C03656=1161.878,20.189,-47.884,-179.949,6.079,149.078
C03657=1161.873,20.439,-47.898,-179.947,6.081,149.077
C03658=1161.869,20.689,-47.912,-179.944,6.081,149.077
C03659=1161.864,20.939,-47.927,-179.941,6.082,149.076
C03660=1161.859,21.188,-47.941,-179.939,6.082,149.075
C03661=1161.854,21.437,-47.956,-179.936,6.083,149.075
C03662=1161.848,21.686,-47.970,-179.934,6.084,149.074
C03663=1161.843,21.936,-47.984,-179.931,6.085,149.074
C03664=1161.838,22.186,-47.999,-179.929,6.086,149.073
C03665=1161.833,22.436,-48.013,-179.926,6.086,149.072
C03666=1161.828,22.686,-48.028,-179.924,6.087,149.072
C03667=1161.823,22.935,-48.043,-179.921,6.088,149.071
C03668=1161.818,23.184,-48.057,-179.919,6.089,149.071
C03669=1161.813,23.433,-48.071,-179.916,6.090,149.070
C03670=1161.808,23.683,-48.085,-179.914,6.090,149.070
C03671=1161.803,23.933,-48.099,-179.911,6.092,149.069
C03672=1161.797,24.182,-48.115,-179.908,6.093,149.069
C03673=1161.792,24.432,-48.129,-179.906,6.093,149.068
C03674=1161.787,24.682,-48.144,-179.903,6.094,149.067
C03675=1161.783,24.931,-48.158,-179.900,6.095,149.067
C03676=1161.778,25.180,-48.173,-179.898,6.096,149.066
C03677=1161.773,25.430,-48.187,-179.896,6.097,149.066
C03678=1161.767,25.679,-48.202,-179.893,6.097,149.065
C03679=1161.762,25.928,-48.217,-179.891,6.098,149.064
C03680=1161.757,26.178,-48.231,-179.888,6.099,149.064
C03681=1161.752,26.428,-48.245,-179.885,6.100,149.063
C03682=1161.747,26.678,-48.259,-179.883,6.100,149.063
C03683=1161.742,26.927,-48.275,-179.881,6.101,149.062
C03684=1161.737,27.177,-48.289,-179.877,6.103,149.062
C03685=1161.732,27.426,-48.304,-179.875,6.103,149.061
C03686=1161.727,27.695,-48.319,-179.873,6.104,149.060
C03687=1161.721,27.964,-48.336,-179.869,6.105,149.060
C03688=1161.716,28.233,-48.351,-179.867,6.106,149.059
C03689=1161.711,28.502,-48.367,-179.864,6.107,149.059
C03690=1161.705,28.752,-48.382,-179.861,6.108,149.058
C03691=1161.700,29.000,-48.396,-179.859,6.109,149.057
C03692=1161.695,29.250,-48.411,-179.856,6.109,149.057
C03693=1161.690,29.499,-48.426,-179.854,6.111,149.056
C03694=1161.684,29.749,-48.441,-179.851,6.111,149.056
C03695=1161.680,29.998,-48.456,-179.849,6.112,149.055
C03696=1161.675,30.248,-48.470,-179.846,6.112,149.055
C03697=1161.669,30.497,-48.485,-179.843,6.114,149.054
C03698=1161.664,30.747,-48.500,-179.841,6.115,149.053
C03699=1161.659,30.997,-48.514,-179.839,6.115,149.053
C03700=1161.654,31.246,-48.530,-179.836,6.116,149.052
C03701=1161.649,31.496,-48.544,-179.833,6.118,149.052
C03702=1161.644,31.745,-48.559,-179.831,6.118,149.051
C03703=1161.639,31.995,-48.574,-179.828,6.119,149.051
C03704=1161.634,32.244,-48.589,-179.825,6.120,149.050
C03705=1161.629,32.493,-48.604,-179.823,6.121,149.049
C03706=1161.624,32.743,-48.619,-179.820,6.121,149.049
C03707=1161.619,32.992,-48.634,-179.818,6.122,149.048
C03708=1161.614,33.242,-48.648,-179.815,6.124,149.048
C03709=1161.609,33.492,-48.664,-179.812,6.124,149.047
C03710=1161.604,33.742,-48.678,-179.810,6.125,149.047
C03711=1161.599,33.991,-48.694,-179.807,6.126,149.046
C03712=1161.594,34.241,-48.708,-179.805,6.127,149.046
C03713=1161.589,34.490,-48.723,-179.802,6.128,149.045
C03714=1161.584,34.739,-48.739,-179.800,6.128,149.044
C03715=1161.579,34.989,-48.753,-179.797,6.130,149.044
C03716=1161.574,35.239,-48.768,-179.795,6.131,149.043
C03717=1161.569,35.488,-48.783,-179.792,6.131,149.043
C03718=1161.564,35.737,-48.798,-179.789,6.133,149.042
C03719=1161.559,35.987,-48.813,-179.787,6.133,149.041
C03720=1161.554,36.236,-48.828,-179.784,6.134,149.041
C03721=1161.548,36.486,-48.843,-179.782,6.134,149.040
C03722=1161.544,36.735,-48.858,-179.779,6.136,149.040
C03723=1161.538,36.984,-48.874,-179.776,6.137,149.039
C03724=1161.534,37.235,-48.888,-179.774,6.137,149.039
C03725=1161.529,37.484,-48.904,-179.771,6.139,149.038
C03726=1161.524,37.733,-48.919,-179.769,6.140,149.038
C03727=1161.518,37.983,-48.934,-179.766,6.140,149.037
C03728=1161.514,38.232,-48.949,-179.763,6.142,149.037
C03729=1161.508,38.482,-48.964,-179.761,6.142,149.036
C03730=1161.504,38.731,-48.979,-179.759,6.143,149.035
C03731=1161.498,38.981,-48.994,-179.755,6.144,149.035
C03732=1161.493,39.230,-49.009,-179.753,6.145,149.034
C03733=1161.488,39.480,-49.025,-179.751,6.146,149.034
C03734=1161.484,39.729,-49.040,-179.748,6.147,149.033
C03735=1161.478,39.979,-49.056,-179.745,6.148,149.033
C03736=1161.473,40.229,-49.071,-179.743,6.149,149.032
C03737=1161.468,40.478,-49.086,-179.740,6.150,149.031
C03738=1161.463,40.727,-49.101,-179.738,6.151,149.031
C03739=1161.458,40.976,-49.116,-179.735,6.151,149.030
C03740=1161.453,41.226,-49.132,-179.732,6.153,149.030
C03741=1161.449,41.475,-49.147,-179.730,6.153,149.029
C03742=1161.443,41.725,-49.162,-179.727,6.154,149.029
C03743=1161.438,41.975,-49.178,-179.724,6.156,149.028
C03744=1161.433,42.224,-49.193,-179.722,6.156,149.028
C03745=1161.428,42.474,-49.209,-179.719,6.157,149.027
C03746=1161.423,42.723,-49.224,-179.717,6.159,149.026
C03747=1161.418,42.972,-49.239,-179.714,6.159,149.026
C03748=1161.413,43.222,-49.255,-179.712,6.160,149.025
C03749=1161.408,43.471,-49.270,-179.709,6.161,149.025
C03750=1161.403,43.721,-49.286,-179.706,6.162,149.024
C03751=1161.398,43.970,-49.301,-179.704,6.163,149.024
C03752=1161.393,44.220,-49.316,-179.701,6.164,149.023
C03753=1161.388,44.469,-49.332,-179.698,6.165,149.022
C03754=1161.382,44.718,-49.347,-179.696,6.166,149.022
C03755=1161.378,44.968,-49.363,-179.693,6.167,149.021
C03756=1161.373,45.218,-49.378,-179.691,6.168,149.021
C03757=1161.368,45.467,-49.394,-179.688,6.168,149.020
C03758=1161.363,45.716,-49.409,-179.686,6.170,149.020
C03759=1161.358,45.966,-49.425,-179.683,6.171,149.019
C03760=1161.353,46.216,-49.441,-179.680,6.172,149.019
C03761=1161.348,46.465,-49.456,-179.678,6.173,149.018
C03762=1161.343,46.714,-49.471,-179.675,6.173,149.018
C03763=1161.338,46.964,-49.487,-179.673,6.175,149.017
C03764=1161.333,47.214,-49.503,-179.670,6.175,149.016
C03765=1161.328,47.463,-49.518,-179.668,6.176,149.016
C03766=1161.323,47.712,-49.533,-179.665,6.178,149.015
C03767=1161.318,47.962,-49.549,-179.662,6.178,149.015
C03768=1161.312,48.212,-49.565,-179.659,6.180,149.014
C03769=1161.308,48.461,-49.580,-179.657,6.181,149.014
C03770=1161.303,48.710,-49.596,-179.654,6.181,149.013
C03771=1161.298,48.960,-49.612,-179.652,6.183,149.013
C03772=1161.292,49.209,-49.628,-179.649,6.183,149.012
C03773=1161.288,49.459,-49.643,-179.647,6.184,149.012
C03774=1161.283,49.708,-49.659,-179.644,6.185,149.011
C03775=1161.278,49.958,-49.674,-179.641,6.186,149.010
C03776=1161.273,50.207,-49.691,-179.638,6.188,149.010
C03777=1161.268,50.456,-49.706,-179.636,6.188,149.009
C03778=1161.263,50.706,-49.721,-179.633,6.189,149.009
C03779=1161.258,50.956,-49.737,-179.631,6.191,149.008
C03780=1161.253,51.205,-49.753,-179.629,6.191,149.008
C03781=1161.248,51.454,-49.769,-179.625,6.193,149.007
C03782=1161.243,51.704,-49.785,-179.623,6.194,149.007
C03783=1161.238,51.953,-49.801,-179.620,6.194,149.006
C03784=1161.233,52.202,-49.816,-179.618,6.196,149.006
C03785=1161.229,52.452,-49.832,-179.615,6.196,149.005
C03786=1161.223,52.701,-49.848,-179.612,6.198,149.004
C03787=1161.218,52.951,-49.864,-179.610,6.198,149.004
C03788=1161.213,53.201,-49.880,-179.608,6.199,149.003
C03789=1161.208,53.450,-49.896,-179.604,6.201,149.003
C03790=1161.202,53.718,-49.913,-179.602,6.201,149.002
C03791=1161.197,53.987,-49.930,-179.599,6.203,149.002
C03792=1161.192,54.256,-49.947,-179.596,6.204,149.001
C03793=1161.186,54.524,-49.964,-179.594,6.205,149.000
C03794=1161.181,54.774,-49.980,-179.590,6.206,149.000
C03795=1161.176,55.023,-49.997,-179.588,6.207,148.999
C03796=1161.171,55.273,-50.012,-179.586,6.208,148.999
C03797=1161.167,55.522,-50.029,-179.583,6.209,148.998
C03798=1161.161,55.771,-50.044,-179.580,6.210,148.998
C03799=1161.156,56.021,-50.060,-179.577,6.211,148.997
C03800=1161.152,56.270,-50.076,-179.575,6.212,148.997
C03801=1161.147,56.519,-50.092,-179.572,6.213,148.996
C03802=1161.142,56.769,-50.108,-179.570,6.214,148.996
C03803=1161.137,57.018,-50.124,-179.567,6.215,148.995
C03804=1161.132,57.268,-50.140,-179.565,6.217,148.994
C03805=1161.127,57.517,-50.156,-179.562,6.217,148.994
C03806=1161.122,57.767,-50.172,-179.559,6.219,148.993
C03807=1161.117,58.016,-50.188,-179.557,6.219,148.993
C03808=1161.112,58.265,-50.204,-179.554,6.221,148.992
C03809=1161.106,58.515,-50.221,-179.552,6.222,148.992
C03810=1161.101,58.765,-50.237,-179.548,6.223,148.991
C03811=1161.097,59.014,-50.254,-179.546,6.224,148.991
C03812=1161.091,59.264,-50.269,-179.544,6.224,148.990
C03813=1161.087,59.513,-50.286,-179.541,6.226,148.990
C03814=1161.081,59.762,-50.301,-179.538,6.227,148.989
C03815=1161.077,60.012,-50.318,-179.535,6.228,148.989
C03816=1161.072,60.261,-50.334,-179.533,6.229,148.988
C03817=1161.067,60.511,-50.350,-179.530,6.230,148.987
C03818=1161.062,60.760,-50.367,-179.528,6.231,148.987
C03819=1161.057,61.010,-50.383,-179.525,6.233,148.986
C03820=1161.052,61.258,-50.399,-179.523,6.233,148.986
C03821=1161.048,61.508,-50.416,-179.519,6.235,148.985
C03822=1161.041,61.758,-50.432,-179.517,6.236,148.985
C03823=1161.037,62.007,-50.448,-179.514,6.237,148.984
C03824=1161.032,62.257,-50.464,-179.512,6.238,148.984
C03825=1161.027,62.506,-50.481,-179.510,6.239,148.983
C03826=1161.022,62.755,-50.497,-179.506,6.240,148.983
C03827=1161.017,63.005,-50.513,-179.504,6.241,148.982
C03828=1161.013,63.254,-50.530,-179.501,6.242,148.982
C03829=1161.008,63.503,-50.546,-179.499,6.243,148.981
C03830=1161.002,63.753,-50.563,-179.496,6.244,148.980
C03831=1160.997,64.002,-50.579,-179.494,6.245,148.980
C03832=1160.993,64.252,-50.595,-179.491,6.247,148.980
C03833=1160.987,64.501,-50.612,-179.488,6.247,148.979
C03834=1160.983,64.751,-50.628,-179.485,6.249,148.978
C03835=1160.977,65.001,-50.645,-179.483,6.250,148.978
C03836=1160.972,65.249,-50.661,-179.480,6.251,148.977
C03837=1160.968,65.499,-50.678,-179.477,6.252,148.977
C03838=1160.963,65.748,-50.693,-179.475,6.253,148.976
C03839=1160.958,65.998,-50.710,-179.473,6.254,148.976
C03840=1160.953,66.247,-50.727,-179.469,6.256,148.975
C03841=1160.948,66.496,-50.744,-179.467,6.256,148.975
C03842=1160.943,66.746,-50.760,-179.464,6.258,148.974
C03843=1160.938,66.995,-50.777,-179.462,6.259,148.974
C03844=1160.933,67.245,-50.793,-179.459,6.260,148.973
C03845=1160.928,67.494,-50.810,-179.456,6.261,148.973
C03846=1160.923,67.743,-50.826,-179.454,6.262,148.972
C03847=1160.919,67.993,-50.843,-179.451,6.263,148.971
C03848=1160.913,68.242,-50.860,-179.448,6.265,148.971
C03849=1160.908,68.491,-50.876,-179.446,6.265,148.970
C03850=1160.904,68.741,-50.893,-179.443,6.267,148.970
C03851=1160.898,68.990,-50.909,-179.441,6.268,148.970
C03852=1160.893,69.240,-50.926,-179.438,6.269,148.969
C03853=1160.889,69.489,-50.943,-179.435,6.270,148.968
C03854=1160.883,69.739,-50.960,-179.432,6.271,148.968
C03855=1160.878,69.988,-50.976,-179.430,6.272,148.967
C03856=1160.874,70.237,-50.993,-179.427,6.274,148.967
C03857=1160.868,70.487,-51.010,-179.425,6.274,148.966
C03858=1160.864,70.736,-51.026,-179.422,6.276,148.966
C03859=1160.859,70.986,-51.043,-179.419,6.277,148.965
C03860=1160.854,71.235,-51.060,-179.417,6.278,148.965
C03861=1160.849,71.484,-51.077,-179.414,6.280,148.964
C03862=1160.844,71.734,-51.093,-179.411,6.280,148.964
C03863=1160.839,71.983,-51.111,-179.408,6.282,148.963
C03864=1160.834,72.232,-51.127,-179.406,6.282,148.963
C03865=1160.829,72.482,-51.144,-179.403,6.284,148.962
C03866=1160.824,72.731,-51.161,-179.401,6.285,148.962
C03867=1160.819,72.980,-51.177,-179.398,6.286,148.961
C03868=1160.814,73.230,-51.194,-179.396,6.287,148.961
C03869=1160.810,73.480,-51.211,-179.392,6.289,148.960
C03870=1160.804,73.729,-51.228,-179.390,6.289,148.959
C03871=1160.800,73.977,-51.245,-179.387,6.291,148.959
C03872=1160.794,74.227,-51.263,-179.384,6.292,148.958
C03873=1160.790,74.477,-51.279,-179.382,6.293,148.958
C03874=1160.785,74.727,-51.297,-179.379,6.295,148.957
C03875=1160.780,74.975,-51.313,-179.377,6.295,148.957
C03876=1160.774,75.225,-51.330,-179.374,6.297,148.956
C03877=1160.770,75.475,-51.347,-179.371,6.298,148.956
C03878=1160.765,75.724,-51.364,-179.369,6.299,148.955
C03879=1160.760,75.973,-51.381,-179.367,6.300,148.955
C03880=1160.755,76.222,-51.398,-179.363,6.302,148.954
C03881=1160.750,76.472,-51.415,-179.361,6.303,148.954
C03882=1160.745,76.722,-51.432,-179.358,6.304,148.953
C03883=1160.741,76.971,-51.449,-179.355,6.305,148.953
C03884=1160.735,77.220,-51.467,-179.353,6.306,148.952
C03885=1160.731,77.469,-51.483,-179.350,6.308,148.952
C03886=1160.725,77.719,-51.501,-179.348,6.308,148.951
C03887=1160.721,77.968,-51.517,-179.345,6.310,148.951
C03888=1160.716,78.218,-51.535,-179.342,6.311,148.950
C03889=1160.711,78.466,-51.551,-179.340,6.312,148.950
C03890=1160.706,78.716,-51.569,-179.336,6.314,148.949
C03891=1160.701,78.965,-51.587,-179.334,6.315,148.949
C03892=1160.696,79.215,-51.603,-179.331,6.316,148.948
C03893=1160.691,79.465,-51.621,-179.329,6.317,148.948
C03894=1160.686,79.732,-51.638,-179.326,6.318,148.947
C03895=1160.681,80.001,-51.658,-179.323,6.320,148.947
C03896=1160.675,80.270,-51.676,-179.320,6.321,148.946
C03897=1160.670,80.537,-51.694,-179.317,6.323,148.945
C03898=1160.665,80.787,-51.711,-179.315,6.324,148.945
C03899=1160.660,81.036,-51.729,-179.312,6.325,148.944
C03900=1160.655,81.286,-51.746,-179.309,6.326,148.944
C03901=1160.651,81.535,-51.764,-179.307,6.328,148.944
C03902=1160.645,81.785,-51.781,-179.304,6.329,148.943
C03903=1160.641,82.034,-51.798,-179.301,6.330,148.942
C03904=1160.635,82.283,-51.816,-179.299,6.331,148.942
C03905=1160.630,82.533,-51.833,-179.296,6.332,148.941
C03906=1160.626,82.781,-51.850,-179.293,6.334,148.941
C03907=1160.621,83.031,-51.868,-179.291,6.335,148.941
C03908=1160.616,83.280,-51.886,-179.288,6.336,148.940
C03909=1160.611,83.530,-51.903,-179.285,6.338,148.939
C03910=1160.606,83.779,-51.920,-179.283,6.338,148.939
C03911=1160.601,84.029,-51.937,-179.280,6.340,148.938
C03912=1160.596,84.278,-51.955,-179.277,6.341,148.938
C03913=1160.592,84.528,-51.972,-179.274,6.342,148.937
C03914=1160.587,84.777,-51.990,-179.272,6.344,148.937
C03915=1160.582,85.027,-52.007,-179.269,6.345,148.936
C03916=1160.577,85.276,-52.025,-179.266,6.346,148.936
C03917=1160.572,85.524,-52.042,-179.264,6.348,148.935
C03918=1160.567,85.774,-52.060,-179.262,6.348,148.935
C03919=1160.562,86.023,-52.077,-179.258,6.350,148.934
C03920=1160.557,86.273,-52.095,-179.256,6.351,148.934
C03921=1160.552,86.522,-52.113,-179.253,6.352,148.933
C03922=1160.547,86.771,-52.129,-179.250,6.354,148.933
C03923=1160.542,87.020,-52.147,-179.247,6.355,148.932
C03924=1160.537,87.270,-52.165,-179.245,6.356,148.932
C03925=1160.532,87.519,-52.183,-179.242,6.358,148.931
C03926=1160.527,87.769,-52.201,-179.239,6.359,148.931
C03927=1160.523,88.018,-52.217,-179.237,6.360,148.930
C03928=1160.518,88.267,-52.235,-179.234,6.361,148.930
C03929=1160.513,88.516,-52.253,-179.231,6.363,148.929
C03930=1160.508,88.766,-52.271,-179.229,6.364,148.929
C03931=1160.503,89.015,-52.289,-179.226,6.365,148.928
C03932=1160.498,89.265,-52.307,-179.224,6.366,148.928
C03933=1160.493,89.514,-52.325,-179.221,6.368,148.928
C03934=1160.489,89.763,-52.341,-179.218,6.370,148.927
C03935=1160.484,90.012,-52.359,-179.216,6.370,148.926
C03936=1160.479,90.262,-52.377,-179.213,6.372,148.926
C03937=1160.474,90.511,-52.394,-179.210,6.374,148.926
C03938=1160.469,90.761,-52.412,-179.208,6.374,148.925
C03939=1160.464,91.010,-52.430,-179.205,6.376,148.925
C03940=1160.459,91.259,-52.448,-179.202,6.377,148.924
C03941=1160.454,91.509,-52.467,-179.200,6.378,148.923
C03942=1160.449,91.759,-52.484,-179.197,6.380,148.923
C03943=1160.444,92.008,-52.502,-179.194,6.381,148.923
C03944=1160.439,92.257,-52.520,-179.192,6.382,148.922
C03945=1160.435,92.506,-52.538,-179.189,6.384,148.922
C03946=1160.430,92.755,-52.556,-179.186,6.385,148.921
C03947=1160.425,93.004,-52.574,-179.183,6.386,148.920
C03948=1160.421,93.253,-52.591,-179.181,6.387,148.920
C03949=1160.415,93.503,-52.609,-179.178,6.389,148.920
C03950=1160.410,93.752,-52.627,-179.175,6.391,148.919
C03951=1160.405,94.001,-52.644,-179.173,6.391,148.919
C03952=1160.401,94.251,-52.662,-179.170,6.393,148.918
C03953=1160.396,94.501,-52.681,-179.167,6.395,148.918
C03954=1160.391,94.750,-52.699,-179.165,6.395,148.917
C03955=1160.386,94.999,-52.717,-179.162,6.397,148.917
C03956=1160.381,95.248,-52.735,-179.159,6.399,148.916
C03957=1160.376,95.498,-52.753,-179.156,6.399,148.916
C03958=1160.371,95.747,-52.771,-179.154,6.401,148.915
C03959=1160.366,95.996,-52.789,-179.151,6.403,148.915
C03960=1160.361,96.245,-52.807,-179.149,6.403,148.914
C03961=1160.357,96.495,-52.826,-179.146,6.405,148.914
C03962=1160.352,96.744,-52.844,-179.143,6.407,148.913
C03963=1160.347,96.993,-52.862,-179.140,6.408,148.913
C03964=1160.342,97.242,-52.880,-179.138,6.409,148.912
C03965=1160.337,97.492,-52.898,-179.135,6.410,148.912
C03966=1160.332,97.741,-52.916,-179.132,6.412,148.911
C03967=1160.328,97.991,-52.934,-179.130,6.413,148.911
C03968=1160.322,98.240,-52.952,-179.127,6.414,148.910
C03969=1160.317,98.489,-52.970,-179.124,6.416,148.910
C03970=1160.312,98.739,-52.988,-179.121,6.418,148.910
C03971=1160.308,98.988,-53.006,-179.119,6.418,148.909
C03972=1160.303,99.237,-53.024,-179.116,6.420,148.908
C03973=1160.299,99.486,-53.043,-179.113,6.422,148.908
C03974=1160.294,99.735,-53.061,-179.111,6.423,148.908
C03975=1160.288,99.985,-53.080,-179.108,6.424,148.907
C03976=1160.283,100.234,-53.098,-179.105,6.426,148.907
C03977=1160.279,100.484,-53.116,-179.102,6.427,148.906
C03978=1160.274,100.733,-53.134,-179.100,6.428,148.906
C03979=1160.269,100.982,-53.153,-179.097,6.430,148.905
C03980=1160.264,101.231,-53.172,-179.094,6.431,148.905
C03981=1160.259,101.480,-53.190,-179.092,6.433,148.904
C03982=1160.254,101.730,-53.208,-179.090,6.434,148.904
C03983=1160.250,101.979,-53.226,-179.086,6.435,148.903
C03984=1160.245,102.228,-53.245,-179.084,6.437,148.903
C03985=1160.239,102.477,-53.263,-179.081,6.439,148.902
C03986=1160.235,102.727,-53.281,-179.078,6.439,148.902
C03987=1160.230,102.976,-53.299,-179.076,6.441,148.901
C03988=1160.225,103.225,-53.318,-179.073,6.443,148.901
C03989=1160.220,103.475,-53.337,-179.070,6.444,148.901
C03990=1160.216,103.724,-53.355,-179.068,6.445,148.900
C03991=1160.211,103.973,-53.374,-179.065,6.446,148.899
C03992=1160.205,104.222,-53.392,-179.062,6.448,148.899
C03993=1160.201,104.472,-53.411,-179.059,6.450,148.899
C03994=1160.196,104.721,-53.429,-179.057,6.450,148.898
C03995=1160.191,104.970,-53.447,-179.054,6.452,148.898
C03996=1160.186,105.220,-53.466,-179.051,6.454,148.897
C03997=1160.182,105.469,-53.485,-179.049,6.456,148.897
C03998=1160.176,105.737,-53.505,-179.045,6.457,148.896
C03999=1160.171,106.006,-53.524,-179.043,6.459,148.896
C04000=1160.166,106.274,-53.545,-179.040,6.460,148.895
C04001=1160.161,106.542,-53.565,-179.037,6.462,148.895
C04002=1160.155,106.792,-53.583,-179.035,6.463,148.894
C04003=1160.151,107.041,-53.603,-179.032,6.464,148.894
C04004=1160.146,107.290,-53.621,-179.029,6.466,148.893
C04005=1160.141,107.539,-53.640,-179.026,6.467,148.893
C04006=1160.137,107.789,-53.658,-179.023,6.469,148.892
C04007=1160.132,108.038,-53.677,-179.021,6.470,148.892
C04008=1160.126,108.287,-53.695,-179.018,6.471,148.891
C04009=1160.122,108.536,-53.714,-179.015,6.473,148.891
C04010=1160.117,108.786,-53.733,-179.012,6.475,148.891
C04011=1160.112,109.034,-53.752,-179.010,6.476,148.890
C04012=1160.107,109.285,-53.771,-179.008,6.477,148.890
C04013=1160.102,109.533,-53.789,-179.004,6.479,148.889
C04014=1160.098,109.783,-53.808,-179.002,6.480,148.889
C04015=1160.093,110.032,-53.827,-178.999,6.482,148.888
C04016=1160.088,110.281,-53.846,-178.997,6.483,148.888
C04017=1160.083,110.531,-53.865,-178.994,6.484,148.887
C04018=1160.079,110.779,-53.883,-178.991,6.486,148.887
C04019=1160.074,111.029,-53.902,-178.988,6.488,148.886
C04020=1160.069,111.278,-53.921,-178.985,6.489,148.886
C04021=1160.064,111.528,-53.941,-178.983,6.490,148.886
C04022=1160.059,111.777,-53.959,-178.980,6.492,148.885
C04023=1160.054,112.026,-53.978,-178.977,6.493,148.885
C04024=1160.050,112.275,-53.997,-178.975,6.495,148.884
C04025=1160.044,112.524,-54.016,-178.972,6.497,148.884
C04026=1160.040,112.774,-54.035,-178.969,6.498,148.883
C04027=1160.035,113.022,-54.054,-178.967,6.499,148.883
C04028=1160.030,113.273,-54.073,-178.964,6.501,148.882
C04029=1160.025,113.521,-54.092,-178.961,6.502,148.882
C04030=1160.021,113.771,-54.111,-178.958,6.504,148.882
C04031=1160.016,114.020,-54.129,-178.956,6.506,148.881
C04032=1160.010,114.269,-54.148,-178.953,6.507,148.880
C04033=1160.006,114.518,-54.168,-178.950,6.508,148.880
C04034=1160.001,114.767,-54.187,-178.948,6.510,148.880
C04035=1159.996,115.017,-54.206,-178.945,6.511,148.879
C04036=1159.991,115.266,-54.224,-178.942,6.513,148.879
C04037=1159.987,115.515,-54.244,-178.939,6.515,148.878
C04038=1159.981,115.764,-54.263,-178.936,6.516,148.878
C04039=1159.977,116.013,-54.282,-178.934,6.517,148.877
C04040=1159.972,116.262,-54.302,-178.932,6.519,148.877
C04041=1159.968,116.512,-54.320,-178.929,6.521,148.877
C04042=1159.962,116.761,-54.339,-178.926,6.522,148.876
C04043=1159.957,117.011,-54.359,-178.923,6.524,148.876
C04044=1159.953,117.260,-54.378,-178.920,6.525,148.875
C04045=1159.948,117.509,-54.397,-178.918,6.526,148.875
C04046=1159.943,117.758,-54.417,-178.915,6.528,148.874
C04047=1159.939,118.007,-54.436,-178.913,6.530,148.874
C04048=1159.934,118.256,-54.455,-178.910,6.531,148.874
C04049=1159.929,118.505,-54.475,-178.907,6.533,148.873
C04050=1159.924,118.755,-54.494,-178.904,6.534,148.873
C04051=1159.919,119.004,-54.512,-178.901,6.536,148.872
C04052=1159.914,119.254,-54.532,-178.899,6.538,148.872
C04053=1159.910,119.503,-54.552,-178.896,6.539,148.871
C04054=1159.904,119.752,-54.571,-178.894,6.541,148.871
C04055=1159.900,120.001,-54.590,-178.891,6.542,148.870
C04056=1159.895,120.250,-54.609,-178.888,6.544,148.870
C04057=1159.890,120.500,-54.629,-178.885,6.545,148.870
C04058=1159.885,120.749,-54.648,-178.882,6.547,148.869
C04059=1159.881,120.998,-54.667,-178.880,6.549,148.869
C04060=1159.876,121.247,-54.687,-178.878,6.550,148.868
C04061=1159.871,121.496,-54.706,-178.874,6.551,148.868
C04062=1159.866,121.745,-54.727,-178.872,6.553,148.867
C04063=1159.862,121.994,-54.746,-178.869,6.554,148.867
C04064=1159.857,122.243,-54.765,-178.866,6.556,148.866
C04065=1159.852,122.493,-54.785,-178.863,6.558,148.866
C04066=1159.847,122.742,-54.804,-178.861,6.560,148.866
C04067=1159.842,122.991,-54.824,-178.858,6.561,148.865
C04068=1159.837,123.241,-54.843,-178.855,6.563,148.865
C04069=1159.833,123.489,-54.862,-178.853,6.564,148.864
C04070=1159.828,123.739,-54.882,-178.850,6.565,148.864
C04071=1159.823,123.988,-54.902,-178.847,6.567,148.863
C04072=1159.818,124.237,-54.921,-178.845,6.569,148.863
C04073=1159.813,124.486,-54.941,-178.842,6.570,148.863
C04074=1159.809,124.736,-54.961,-178.839,6.572,148.862
C04075=1159.803,124.985,-54.980,-178.836,6.573,148.862
C04076=1159.799,125.234,-55.000,-178.833,6.575,148.861
C04077=1159.794,125.483,-55.020,-178.831,6.577,148.861
C04078=1159.790,125.732,-55.039,-178.828,6.579,148.860
C04079=1159.785,125.981,-55.058,-178.825,6.580,148.860
C04080=1159.780,126.230,-55.079,-178.823,6.581,148.860
C04081=1159.776,126.480,-55.098,-178.820,6.583,148.859
C04082=1159.770,126.729,-55.118,-178.818,6.585,148.859
C04083=1159.766,126.978,-55.137,-178.814,6.586,148.858
C04084=1159.761,127.227,-55.158,-178.812,6.588,148.858
C04085=1159.756,127.477,-55.177,-178.809,6.589,148.857
C04086=1159.751,127.726,-55.197,-178.806,6.591,148.857
C04087=1159.747,127.975,-55.217,-178.804,6.593,148.857
C04088=1159.742,128.224,-55.237,-178.801,6.595,148.856
C04089=1159.737,128.474,-55.256,-178.798,6.596,148.856
C04090=1159.732,128.722,-55.276,-178.795,6.598,148.855
C04091=1159.727,128.972,-55.296,-178.793,6.600,148.855
C04092=1159.723,129.221,-55.316,-178.789,6.601,148.854
C04093=1159.718,129.470,-55.336,-178.787,6.603,148.854
C04094=1159.713,129.719,-55.355,-178.785,6.604,148.854
C04095=1159.708,129.968,-55.376,-178.782,6.606,148.853
C04096=1159.704,130.218,-55.395,-178.779,6.607,148.853
C04097=1159.699,130.467,-55.416,-178.777,6.609,148.852
C04098=1159.694,130.715,-55.435,-178.774,6.611,148.852
C04099=1159.689,130.964,-55.455,-178.771,6.612,148.852
C04100=1159.685,131.214,-55.475,-178.768,6.614,148.851
C04101=1159.679,131.463,-55.496,-178.766,6.616,148.851
C04102=1159.675,131.732,-55.517,-178.762,6.617,148.850
C04103=1159.670,132.001,-55.538,-178.759,6.620,148.850
C04104=1159.664,132.269,-55.560,-178.756,6.621,148.849
C04105=1159.659,132.538,-55.582,-178.754,6.623,148.849
C04106=1159.655,132.786,-55.602,-178.751,6.625,148.849
C04107=1159.649,133.036,-55.622,-178.748,6.626,148.848
C04108=1159.644,133.285,-55.642,-178.745,6.628,148.848
C04109=1159.640,133.534,-55.662,-178.742,6.630,148.847
C04110=1159.635,133.783,-55.682,-178.740,6.631,148.847
C04111=1159.630,134.033,-55.702,-178.737,6.633,148.847
C04112=1159.626,134.282,-55.722,-178.734,6.635,148.846
C04113=1159.620,134.530,-55.743,-178.732,6.637,148.846
C04114=1159.616,134.780,-55.762,-178.729,6.638,148.845
C04115=1159.611,135.029,-55.783,-178.726,6.640,148.845
C04116=1159.607,135.278,-55.803,-178.723,6.642,148.845
C04117=1159.602,135.527,-55.823,-178.721,6.644,148.844
C04118=1159.597,135.776,-55.844,-178.718,6.645,148.844
C04119=1159.592,136.025,-55.864,-178.715,6.647,148.843
C04120=1159.588,136.275,-55.884,-178.713,6.649,148.843
C04121=1159.583,136.524,-55.904,-178.710,6.650,148.843
C04122=1159.577,136.773,-55.925,-178.707,6.652,148.842
C04123=1159.573,137.021,-55.945,-178.704,6.654,148.842
C04124=1159.568,137.271,-55.965,-178.701,6.655,148.841
C04125=1159.564,137.520,-55.985,-178.699,6.657,148.841
C04126=1159.559,137.769,-56.006,-178.696,6.659,148.840
C04127=1159.554,138.018,-56.027,-178.693,6.660,148.840
C04128=1159.549,138.268,-56.046,-178.691,6.662,148.840
C04129=1159.545,138.517,-56.067,-178.688,6.664,148.839
C04130=1159.540,138.766,-56.088,-178.685,6.666,148.839
C04131=1159.535,139.015,-56.108,-178.682,6.667,148.839
C04132=1159.531,139.264,-56.128,-178.680,6.669,148.838
C04133=1159.525,139.514,-56.149,-178.677,6.671,148.838
C04134=1159.521,139.763,-56.169,-178.674,6.672,148.837
C04135=1159.517,140.012,-56.189,-178.672,6.674,148.837
C04136=1159.511,140.261,-56.210,-178.669,6.676,148.837
C04137=1159.507,140.510,-56.231,-178.666,6.678,148.836
C04138=1159.502,140.759,-56.251,-178.663,6.679,148.836
C04139=1159.497,141.008,-56.272,-178.661,6.681,148.835
C04140=1159.493,141.257,-56.292,-178.658,6.683,148.835
C04141=1159.488,141.506,-56.313,-178.655,6.685,148.835
C04142=1159.483,141.755,-56.334,-178.653,6.686,148.834
C04143=1159.479,142.004,-56.354,-178.650,6.688,148.834
C04144=1159.474,142.253,-56.375,-178.647,6.690,148.833
C04145=1159.469,142.502,-56.395,-178.645,6.692,148.833
C04146=1159.464,142.752,-56.416,-178.642,6.693,148.833
C04147=1159.460,143.001,-56.437,-178.639,6.695,148.832
C04148=1159.454,143.250,-56.458,-178.636,6.697,148.832
C04149=1159.450,143.499,-56.478,-178.634,6.698,148.832
C04150=1159.446,143.748,-56.498,-178.631,6.700,148.831
C04151=1159.440,143.997,-56.519,-178.628,6.702,148.831
C04152=1159.436,144.246,-56.540,-178.626,6.704,148.830
C04153=1159.431,144.495,-56.561,-178.623,6.705,148.830
C04154=1159.426,144.744,-56.581,-178.620,6.707,148.830
C04155=1159.421,144.993,-56.602,-178.617,6.709,148.829
C04156=1159.417,145.242,-56.622,-178.615,6.711,148.829
C04157=1159.412,145.492,-56.643,-178.612,6.712,148.828
C04158=1159.407,145.741,-56.664,-178.609,6.714,148.828
C04159=1159.402,145.990,-56.685,-178.606,6.717,148.828
C04160=1159.398,146.239,-56.706,-178.603,6.718,148.827
C04161=1159.393,146.488,-56.727,-178.601,6.720,148.827
C04162=1159.389,146.737,-56.748,-178.598,6.722,148.827
C04163=1159.384,146.986,-56.769,-178.595,6.723,148.826
C04164=1159.378,147.236,-56.789,-178.593,6.725,148.826
C04165=1159.374,147.485,-56.810,-178.590,6.727,148.825
C04166=1159.369,147.733,-56.832,-178.587,6.729,148.825
C04167=1159.365,147.982,-56.852,-178.584,6.730,148.825
C04168=1159.360,148.231,-56.873,-178.582,6.732,148.824
C04169=1159.355,148.481,-56.894,-178.579,6.734,148.824
C04170=1159.351,148.730,-56.915,-178.576,6.736,148.823
C04171=1159.346,148.979,-56.936,-178.574,6.737,148.823
C04172=1159.341,149.228,-56.957,-178.571,6.739,148.823
C04173=1159.336,149.477,-56.978,-178.568,6.742,148.822
C04174=1159.331,149.726,-56.999,-178.565,6.743,148.822
C04175=1159.327,149.975,-57.020,-178.562,6.745,148.822
C04176=1159.322,150.225,-57.041,-178.560,6.747,148.821
C04177=1159.317,150.473,-57.063,-178.557,6.749,148.821
C04178=1159.313,150.722,-57.083,-178.554,6.750,148.820
C04179=1159.308,150.971,-57.105,-178.551,6.752,148.820
C04180=1159.303,151.220,-57.126,-178.549,6.754,148.820
C04181=1159.299,151.470,-57.146,-178.546,6.755,148.819
C04182=1159.294,151.718,-57.168,-178.543,6.757,148.819
C04183=1159.289,151.968,-57.189,-178.540,6.760,148.819
C04184=1159.284,152.217,-57.210,-178.537,6.761,148.818
C04185=1159.280,152.465,-57.231,-178.535,6.763,148.818
C04186=1159.275,152.715,-57.252,-178.532,6.765,148.817
C04187=1159.270,152.964,-57.274,-178.530,6.767,148.817
C04188=1159.265,153.213,-57.295,-178.527,6.769,148.817
C04189=1159.261,153.461,-57.316,-178.524,6.771,148.816
C04190=1159.256,153.711,-57.337,-178.522,6.772,148.816
C04191=1159.251,153.960,-57.359,-178.519,6.774,148.816
C04192=1159.246,154.209,-57.380,-178.516,6.777,148.815
C04193=1159.242,154.458,-57.401,-178.513,6.778,148.815
C04194=1159.237,154.707,-57.422,-178.510,6.780,148.815
C04195=1159.233,154.956,-57.444,-178.508,6.782,148.814
C04196=1159.227,155.206,-57.465,-178.505,6.783,148.814
C04197=1159.223,155.454,-57.487,-178.502,6.785,148.813
C04198=1159.218,155.703,-57.508,-178.499,6.787,148.813
C04199=1159.214,155.952,-57.529,-178.497,6.789,148.813
C04200=1159.209,156.201,-57.551,-178.493,6.791,148.812
C04201=1159.204,156.450,-57.572,-178.491,6.793,148.812
C04202=1159.200,156.700,-57.594,-178.489,6.795,148.812
C04203=1159.195,156.948,-57.616,-178.486,6.797,148.811
C04204=1159.190,157.198,-57.637,-178.483,6.799,148.811
C04205=1159.186,157.447,-57.658,-178.480,6.800,148.811
C04206=1159.180,157.715,-57.681,-178.477,6.803,148.810
C04207=1159.175,157.984,-57.704,-178.474,6.805,148.810
C04208=1159.170,158.253,-57.728,-178.471,6.807,148.810
C04209=1159.165,158.522,-57.751,-178.468,6.809,148.809
C04210=1159.161,158.771,-57.773,-178.466,6.811,148.809
C04211=1159.156,159.021,-57.794,-178.463,6.812,148.808
C04212=1159.151,159.269,-57.815,-178.460,6.814,148.808
C04213=1159.147,159.519,-57.838,-178.457,6.817,148.808
C04214=1159.142,159.767,-57.859,-178.454,6.818,148.807
C04215=1159.137,160.016,-57.881,-178.452,6.820,148.807
C04216=1159.132,160.266,-57.902,-178.449,6.822,148.807
C04217=1159.128,160.515,-57.924,-178.446,6.824,148.806
C04218=1159.123,160.763,-57.946,-178.444,6.826,148.806
C04219=1159.118,161.013,-57.968,-178.441,6.828,148.806
C04220=1159.113,161.261,-57.989,-178.438,6.830,148.805
C04221=1159.109,161.511,-58.011,-178.435,6.832,148.805
C04222=1159.104,161.760,-58.032,-178.433,6.833,148.805
C04223=1159.099,162.008,-58.054,-178.430,6.835,148.804
C04224=1159.095,162.258,-58.076,-178.427,6.837,148.804
C04225=1159.090,162.506,-58.098,-178.424,6.840,148.804
C04226=1159.086,162.756,-58.120,-178.422,6.842,148.803
C04227=1159.081,163.004,-58.141,-178.419,6.843,148.803
C04228=1159.077,163.254,-58.164,-178.416,6.845,148.803
C04229=1159.072,163.502,-58.185,-178.414,6.847,148.802
C04230=1159.067,163.751,-58.207,-178.410,6.849,148.802
C04231=1159.063,164.000,-58.229,-178.408,6.851,148.802
C04232=1159.057,164.250,-58.250,-178.405,6.853,148.801
C04233=1159.052,164.499,-58.273,-178.403,6.855,148.801
C04234=1159.048,164.748,-58.294,-178.400,6.857,148.801
C04235=1159.043,164.997,-58.316,-178.397,6.859,148.800
C04236=1159.039,165.245,-58.339,-178.394,6.861,148.800
C04237=1159.034,165.495,-58.361,-178.392,6.863,148.800
C04238=1159.030,165.743,-58.382,-178.389,6.864,148.799
C04239=1159.025,165.993,-58.404,-178.386,6.866,148.799
C04240=1159.020,166.241,-58.426,-178.383,6.869,148.799
C04241=1159.015,166.491,-58.449,-178.381,6.871,148.798
C04242=1159.011,166.740,-58.470,-178.378,6.873,148.798
C04243=1159.006,166.989,-58.492,-178.375,6.874,148.798
C04244=1159.001,167.238,-58.514,-178.373,6.876,148.797
C04245=1158.997,167.487,-58.536,-178.369,6.879,148.797
C04246=1158.992,167.736,-58.559,-178.367,6.881,148.797
C04247=1158.987,167.985,-58.581,-178.364,6.883,148.796
C04248=1158.983,168.233,-58.603,-178.362,6.884,148.796
C04249=1158.978,168.483,-58.625,-178.358,6.887,148.796
C04250=1158.974,168.731,-58.647,-178.356,6.889,148.795
C04251=1158.969,168.981,-58.669,-178.353,6.890,148.795
C04252=1158.964,169.229,-58.691,-178.351,6.892,148.795
C04253=1158.960,169.478,-58.714,-178.348,6.894,148.794
C04254=1158.955,169.727,-58.735,-178.345,6.897,148.794
C04255=1158.950,169.976,-58.758,-178.342,6.898,148.794
C04256=1158.945,170.225,-58.780,-178.339,6.900,148.793
C04257=1158.941,170.474,-58.803,-178.337,6.902,148.793
C04258=1158.936,170.724,-58.825,-178.334,6.905,148.793
C04259=1158.931,170.972,-58.847,-178.331,6.907,148.792
C04260=1158.927,171.221,-58.869,-178.329,6.908,148.792
C04261=1158.922,171.470,-58.892,-178.326,6.910,148.792
C04262=1158.917,171.719,-58.914,-178.323,6.913,148.792
C04263=1158.913,171.969,-58.936,-178.320,6.915,148.791
C04264=1158.908,172.217,-58.959,-178.318,6.917,148.791
C04265=1158.904,172.466,-58.981,-178.315,6.918,148.790
C04266=1158.899,172.715,-59.003,-178.312,6.921,148.790
C04267=1158.894,172.964,-59.026,-178.310,6.923,148.790
C04268=1158.890,173.213,-59.048,-178.307,6.925,148.790
C04269=1158.885,173.461,-59.071,-178.304,6.926,148.789
C04270=1158.880,173.711,-59.093,-178.301,6.929,148.789
C04271=1158.875,173.959,-59.115,-178.298,6.931,148.788
C04272=1158.871,174.209,-59.138,-178.296,6.933,148.788
C04273=1158.866,174.458,-59.160,-178.293,6.935,148.788
C04274=1158.862,174.706,-59.183,-178.290,6.937,148.788
C04275=1158.857,174.956,-59.205,-178.287,6.939,148.787
C04276=1158.853,175.204,-59.228,-178.285,6.941,148.787
C04277=1158.847,175.453,-59.250,-178.282,6.944,148.787
C04278=1158.843,175.702,-59.273,-178.279,6.945,148.786
C04279=1158.838,175.952,-59.296,-178.276,6.947,148.786
C04280=1158.834,176.200,-59.318,-178.273,6.950,148.786
C04281=1158.829,176.449,-59.341,-178.271,6.952,148.786
C04282=1158.825,176.698,-59.364,-178.268,6.953,148.785
C04283=1158.820,176.948,-59.386,-178.266,6.955,148.785
C04284=1158.815,177.196,-59.409,-178.262,6.958,148.784
C04285=1158.810,177.445,-59.432,-178.260,6.960,148.784
C04286=1158.806,177.694,-59.454,-178.257,6.962,148.784
C04287=1158.801,177.942,-59.477,-178.254,6.964,148.784
C04288=1158.797,178.191,-59.500,-178.251,6.966,148.783
C04289=1158.792,178.441,-59.522,-178.249,6.968,148.783
C04290=1158.788,178.689,-59.545,-178.247,6.970,148.783
C04291=1158.782,178.938,-59.567,-178.243,6.972,148.782
C04292=1158.778,179.187,-59.590,-178.241,6.974,148.782
C04293=1158.774,179.436,-59.614,-178.238,6.976,148.782
C04294=1158.770,179.685,-59.636,-178.235,6.979,148.782
C04295=1158.764,179.934,-59.659,-178.232,6.981,148.781
C04296=1158.759,180.183,-59.682,-178.230,6.982,148.781
C04297=1158.755,180.432,-59.705,-178.227,6.985,148.781
C04298=1158.750,180.681,-59.727,-178.224,6.987,148.780
C04299=1158.746,180.929,-59.750,-178.222,6.989,148.780
C04300=1158.741,181.178,-59.773,-178.219,6.992,148.780
C04301=1158.736,181.427,-59.796,-178.216,6.993,148.780
C04302=1158.732,181.676,-59.819,-178.213,6.995,148.779
C04303=1158.727,181.926,-59.842,-178.210,6.998,148.779
C04304=1158.722,182.174,-59.865,-178.208,7.000,148.779
C04305=1158.718,182.423,-59.888,-178.205,7.002,148.778
C04306=1158.713,182.672,-59.911,-178.202,7.004,148.778
C04307=1158.709,182.921,-59.934,-178.200,7.006,148.778
C04308=1158.705,183.170,-59.957,-178.197,7.008,148.777
C04309=1158.700,183.419,-59.980,-178.194,7.011,148.777
C04310=1158.695,183.688,-60.006,-178.191,7.012,148.777
C04311=1158.690,183.958,-60.030,-178.188,7.015,148.776
C04312=1158.685,184.228,-60.055,-178.186,7.017,148.776
C04313=1158.680,184.497,-60.080,-178.182,7.020,148.776
C04314=1158.676,184.746,-60.103,-178.180,7.021,148.776
C04315=1158.671,184.995,-60.126,-178.176,7.024,148.775
C04316=1158.666,185.243,-60.149,-178.174,7.026,148.775
C04317=1158.661,185.492,-60.173,-178.172,7.028,148.775
C04318=1158.657,185.741,-60.195,-178.168,7.030,148.774
C04319=1158.652,185.990,-60.219,-178.166,7.032,148.774
C04320=1158.648,186.239,-60.242,-178.163,7.035,148.774
C04321=1158.643,186.488,-60.265,-178.160,7.037,148.774
C04322=1158.638,186.737,-60.289,-178.158,7.039,148.773
C04323=1158.634,186.986,-60.311,-178.155,7.041,148.773
C04324=1158.630,187.235,-60.335,-178.152,7.043,148.773
C04325=1158.624,187.483,-60.358,-178.150,7.045,148.773
C04326=1158.620,187.732,-60.381,-178.146,7.048,148.772
C04327=1158.615,187.981,-60.405,-178.144,7.050,148.772
C04328=1158.610,188.230,-60.428,-178.142,7.052,148.772
C04329=1158.606,188.479,-60.451,-178.138,7.054,148.771
C04330=1158.602,188.728,-60.475,-178.136,7.056,148.771
C04331=1158.597,188.977,-60.498,-178.133,7.059,148.771
C04332=1158.592,189.226,-60.521,-178.130,7.061,148.771
C04333=1158.588,189.475,-60.545,-178.127,7.062,148.770
C04334=1158.583,189.724,-60.568,-178.125,7.065,148.770
C04335=1158.579,189.972,-60.592,-178.122,7.067,148.770
C04336=1158.574,190.221,-60.616,-178.119,7.070,148.769
C04337=1158.569,190.470,-60.639,-178.116,7.072,148.769
C04338=1158.564,190.719,-60.662,-178.114,7.074,148.769
C04339=1158.560,190.968,-60.686,-178.111,7.076,148.769
C04340=1158.555,191.217,-60.710,-178.108,7.078,148.769
C04341=1158.551,191.466,-60.733,-178.105,7.081,148.768
C04342=1158.547,191.714,-60.756,-178.102,7.083,148.768
C04343=1158.542,191.963,-60.780,-178.100,7.085,148.768
C04344=1158.538,192.212,-60.803,-178.097,7.087,148.767
C04345=1158.533,192.461,-60.827,-178.095,7.089,148.767
C04346=1158.528,192.710,-60.850,-178.091,7.092,148.767
C04347=1158.524,192.958,-60.874,-178.089,7.094,148.767
C04348=1158.519,193.207,-60.897,-178.087,7.096,148.766
C04349=1158.514,193.457,-60.921,-178.083,7.098,148.766
C04350=1158.509,193.705,-60.946,-178.081,7.100,148.766
C04351=1158.505,193.954,-60.969,-178.078,7.103,148.766
C04352=1158.500,194.203,-60.993,-178.075,7.105,148.765
C04353=1158.495,194.452,-61.016,-178.073,7.107,148.765
C04354=1158.491,194.701,-61.040,-178.070,7.109,148.765
C04355=1158.486,194.949,-61.064,-178.067,7.111,148.764
C04356=1158.482,195.198,-61.087,-178.064,7.114,148.764
C04357=1158.477,195.447,-61.111,-178.062,7.116,148.764
C04358=1158.473,195.696,-61.135,-178.059,7.119,148.764
C04359=1158.468,195.944,-61.159,-178.056,7.121,148.764
C04360=1158.464,196.193,-61.182,-178.053,7.122,148.763
C04361=1158.460,196.442,-61.206,-178.051,7.125,148.763
C04362=1158.454,196.691,-61.230,-178.048,7.127,148.763
C04363=1158.450,196.940,-61.254,-178.045,7.130,148.763
C04364=1158.445,197.189,-61.278,-178.042,7.132,148.762
C04365=1158.441,197.437,-61.302,-178.039,7.134,148.762
C04366=1158.436,197.686,-61.326,-178.037,7.136,148.762
C04367=1158.432,197.935,-61.349,-178.034,7.139,148.761
C04368=1158.427,198.183,-61.373,-178.031,7.141,148.761
C04369=1158.422,198.433,-61.397,-178.029,7.143,148.761
C04370=1158.418,198.682,-61.422,-178.026,7.146,148.761
C04371=1158.414,198.930,-61.446,-178.023,7.148,148.761
C04372=1158.409,199.179,-61.469,-178.020,7.150,148.760
C04373=1158.405,199.427,-61.493,-178.018,7.152,148.760
C04374=1158.399,199.677,-61.517,-178.015,7.155,148.760
C04375=1158.395,199.925,-61.541,-178.012,7.157,148.760
C04376=1158.391,200.174,-61.566,-178.009,7.160,148.759
C04377=1158.387,200.423,-61.590,-178.007,7.162,148.759
C04378=1158.381,200.672,-61.614,-178.004,7.164,148.759
C04379=1158.377,200.921,-61.638,-178.001,7.166,148.759
C04380=1158.372,201.169,-61.662,-177.998,7.169,148.758
C04381=1158.369,201.418,-61.686,-177.996,7.171,148.758
C04382=1158.363,201.667,-61.710,-177.993,7.173,148.758
C04383=1158.359,201.916,-61.734,-177.990,7.175,148.758
C04384=1158.354,202.164,-61.758,-177.988,7.177,148.757
C04385=1158.349,202.413,-61.783,-177.985,7.180,148.757
C04386=1158.345,202.663,-61.807,-177.982,7.182,148.757
C04387=1158.341,202.911,-61.831,-177.979,7.185,148.757
C04388=1158.336,203.160,-61.856,-177.977,7.187,148.757
C04389=1158.331,203.408,-61.880,-177.974,7.189,148.756
C04390=1158.327,203.657,-61.904,-177.971,7.192,148.756
C04391=1158.322,203.906,-61.929,-177.968,7.194,148.756
C04392=1158.318,204.154,-61.953,-177.966,7.196,148.756
C04393=1158.313,204.403,-61.977,-177.963,7.199,148.755
C04394=1158.309,204.653,-62.001,-177.960,7.201,148.755
C04395=1158.304,204.901,-62.025,-177.957,7.203,148.755
C04396=1158.299,205.150,-62.050,-177.955,7.205,148.755
C04397=1158.295,205.398,-62.074,-177.952,7.208,148.754
C04398=1158.291,205.648,-62.099,-177.949,7.210,148.754
C04399=1158.286,205.896,-62.123,-177.946,7.213,148.754
C04400=1158.281,206.145,-62.147,-177.944,7.215,148.754
C04401=1158.277,206.394,-62.172,-177.941,7.218,148.754
C04402=1158.272,206.643,-62.196,-177.938,7.219,148.753
C04403=1158.267,206.891,-62.221,-177.935,7.222,148.753
C04404=1158.263,207.140,-62.245,-177.933,7.224,148.753
C04405=1158.258,207.389,-62.270,-177.930,7.227,148.753
C04406=1158.254,207.638,-62.294,-177.927,7.229,148.752
C04407=1158.249,207.886,-62.319,-177.925,7.232,148.752
C04408=1158.245,208.135,-62.343,-177.922,7.233,148.752
C04409=1158.240,208.383,-62.369,-177.919,7.236,148.752
C04410=1158.236,208.632,-62.393,-177.916,7.239,148.751
C04411=1158.231,208.881,-62.418,-177.914,7.241,148.751
C04412=1158.227,209.130,-62.442,-177.910,7.244,148.751
C04413=1158.222,209.379,-62.467,-177.908,7.246,148.751
C04414=1158.217,209.649,-62.494,-177.905,7.248,148.751
C04415=1158.212,209.919,-62.520,-177.902,7.251,148.750
C04416=1158.208,210.190,-62.547,-177.899,7.254,148.750
C04417=1158.202,210.461,-62.574,-177.896,7.257,148.750
C04418=1158.199,210.710,-62.599,-177.893,7.259,148.750
C04419=1158.193,210.958,-62.623,-177.891,7.261,148.750
C04420=1158.188,211.207,-62.648,-177.888,7.263,148.749
C04421=1158.185,211.456,-62.673,-177.885,7.266,148.749
C04422=1158.180,211.704,-62.698,-177.882,7.268,148.749
C04423=1158.175,211.954,-62.723,-177.880,7.271,148.749
C04424=1158.171,212.202,-62.748,-177.877,7.273,148.748
C04425=1158.166,212.450,-62.772,-177.874,7.276,148.748
C04426=1158.162,212.699,-62.797,-177.872,7.278,148.748
C04427=1158.157,212.948,-62.821,-177.869,7.280,148.748
C04428=1158.153,213.197,-62.847,-177.866,7.283,148.748
C04429=1158.148,213.445,-62.871,-177.863,7.285,148.747
C04430=1158.144,213.694,-62.897,-177.861,7.288,148.747
C04431=1158.139,213.943,-62.922,-177.858,7.290,148.747
C04432=1158.135,214.192,-62.947,-177.855,7.293,148.747
C04433=1158.130,214.440,-62.971,-177.852,7.294,148.747
C04434=1158.126,214.689,-62.996,-177.850,7.297,148.746
C04435=1158.121,214.938,-63.022,-177.847,7.300,148.746
C04436=1158.117,215.187,-63.046,-177.844,7.302,148.746
C04437=1158.112,215.435,-63.071,-177.841,7.305,148.746
C04438=1158.107,215.684,-63.096,-177.839,7.307,148.746
C04439=1158.103,215.933,-63.121,-177.836,7.310,148.746
C04440=1158.099,216.181,-63.146,-177.833,7.311,148.745
C04441=1158.094,216.430,-63.171,-177.830,7.314,148.745
C04442=1158.090,216.679,-63.197,-177.828,7.317,148.745
C04443=1158.085,216.928,-63.222,-177.825,7.319,148.745
C04444=1158.081,217.177,-63.247,-177.822,7.322,148.745
C04445=1158.077,217.424,-63.272,-177.820,7.324,148.744
C04446=1158.072,217.674,-63.297,-177.817,7.327,148.744
C04447=1158.067,217.922,-63.323,-177.814,7.330,148.744
C04448=1158.063,218.171,-63.348,-177.811,7.331,148.744
C04449=1158.058,218.419,-63.373,-177.809,7.334,148.744
C04450=1158.053,218.669,-63.398,-177.806,7.336,148.743
C04451=1158.049,218.917,-63.423,-177.803,7.339,148.743
C04452=1158.045,219.165,-63.449,-177.800,7.342,148.743
C04453=1158.040,219.415,-63.474,-177.798,7.344,148.743
C04454=1158.036,219.663,-63.499,-177.795,7.347,148.743
C04455=1158.031,219.912,-63.525,-177.793,7.349,148.743
C04456=1158.026,220.160,-63.549,-177.789,7.351,148.742
C04457=1158.022,220.409,-63.575,-177.787,7.354,148.742
C04458=1158.018,220.658,-63.601,-177.784,7.356,148.742
C04459=1158.014,220.906,-63.626,-177.781,7.359,148.742
C04460=1158.009,221.155,-63.651,-177.778,7.362,148.742
C04461=1158.004,221.403,-63.676,-177.776,7.364,148.741
C04462=1158.000,221.652,-63.702,-177.773,7.367,148.741
C04463=1157.996,221.901,-63.728,-177.771,7.369,148.741
C04464=1157.991,222.150,-63.752,-177.768,7.371,148.741
C04465=1157.987,222.398,-63.778,-177.765,7.374,148.741
C04466=1157.982,222.647,-63.803,-177.762,7.376,148.740
C04467=1157.978,222.895,-63.829,-177.759,7.379,148.740
C04468=1157.973,223.144,-63.855,-177.757,7.382,148.740
C04469=1157.968,223.392,-63.880,-177.754,7.384,148.740
C04470=1157.964,223.642,-63.905,-177.751,7.387,148.740
C04471=1157.960,223.891,-63.931,-177.748,7.390,148.740
C04472=1157.955,224.139,-63.956,-177.746,7.391,148.739
C04473=1157.951,224.387,-63.982,-177.743,7.394,148.739
C04474=1157.946,224.636,-64.008,-177.740,7.397,148.739
C04475=1157.942,224.884,-64.033,-177.737,7.399,148.739
C04476=1157.937,225.133,-64.060,-177.735,7.402,148.739
C04477=1157.932,225.382,-64.085,-177.732,7.405,148.739
C04478=1157.928,225.630,-64.111,-177.729,7.407,148.738
C04479=1157.923,225.879,-64.137,-177.726,7.410,148.738
C04480=1157.919,226.128,-64.162,-177.724,7.412,148.738
C04481=1157.915,226.377,-64.188,-177.721,7.414,148.738
C04482=1157.910,226.625,-64.213,-177.718,7.417,148.738
C04483=1157.906,226.874,-64.239,-177.715,7.420,148.738
C04484=1157.902,227.123,-64.265,-177.713,7.422,148.737
C04485=1157.897,227.372,-64.291,-177.710,7.425,148.737
C04486=1157.892,227.620,-64.317,-177.707,7.428,148.737
C04487=1157.888,227.869,-64.342,-177.705,7.430,148.737
C04488=1157.883,228.117,-64.368,-177.702,7.432,148.737
C04489=1157.879,228.366,-64.394,-177.699,7.435,148.737
C04490=1157.874,228.614,-64.419,-177.697,7.438,148.737
C04491=1157.870,228.863,-64.446,-177.694,7.440,148.736
C04492=1157.865,229.112,-64.472,-177.691,7.443,148.736
C04493=1157.861,229.360,-64.498,-177.689,7.445,148.736
C04494=1157.856,229.608,-64.523,-177.685,7.448,148.736
C04495=1157.852,229.857,-64.549,-177.683,7.451,148.736
C04496=1157.847,230.106,-64.575,-177.680,7.453,148.736
C04497=1157.843,230.355,-64.602,-177.678,7.456,148.735
C04498=1157.839,230.603,-64.628,-177.674,7.458,148.735
C04499=1157.834,230.851,-64.653,-177.672,7.461,148.735
C04500=1157.829,231.101,-64.679,-177.669,7.463,148.735
C04501=1157.825,231.349,-64.706,-177.666,7.466,148.735
C04502=1157.821,231.598,-64.732,-177.663,7.469,148.735
C04503=1157.816,231.847,-64.758,-177.661,7.471,148.735
C04504=1157.811,232.095,-64.783,-177.658,7.474,148.734
C04505=1157.807,232.343,-64.810,-177.655,7.477,148.734
C04506=1157.802,232.592,-64.836,-177.653,7.479,148.734
C04507=1157.798,232.841,-64.862,-177.650,7.482,148.734
C04508=1157.794,233.089,-64.888,-177.647,7.485,148.734
C04509=1157.789,233.338,-64.915,-177.644,7.487,148.734
C04510=1157.785,233.586,-64.941,-177.642,7.489,148.733
C04511=1157.781,233.834,-64.967,-177.639,7.492,148.733
C04512=1157.776,234.084,-64.993,-177.636,7.495,148.733
C04513=1157.772,234.332,-65.019,-177.633,7.498,148.733
C04514=1157.768,234.581,-65.045,-177.631,7.500,148.733
C04515=1157.763,234.829,-65.072,-177.628,7.503,148.733
C04516=1157.759,235.078,-65.098,-177.625,7.506,148.733
C04517=1157.754,235.326,-65.125,-177.623,7.508,148.732
C04518=1157.749,235.598,-65.153,-177.619,7.511,148.732
C04519=1157.744,235.870,-65.182,-177.617,7.514,148.732
C04520=1157.739,236.142,-65.210,-177.613,7.517,148.732
C04521=1157.734,236.413,-65.240,-177.611,7.520,148.732
C04522=1157.730,236.662,-65.266,-177.608,7.523,148.732
C04523=1157.725,236.911,-65.293,-177.606,7.525,148.732
C04524=1157.722,237.159,-65.319,-177.602,7.527,148.731
C04525=1157.717,237.408,-65.345,-177.600,7.530,148.731
C04526=1157.713,237.656,-65.372,-177.597,7.533,148.731
C04527=1157.708,237.905,-65.398,-177.595,7.535,148.731
C04528=1157.704,238.153,-65.425,-177.592,7.538,148.731
C04529=1157.699,238.402,-65.452,-177.589,7.541,148.731
C04530=1157.695,238.651,-65.477,-177.586,7.544,148.731
C04531=1157.690,238.899,-65.505,-177.584,7.546,148.731
C04532=1157.686,239.147,-65.531,-177.581,7.549,148.731
C04533=1157.681,239.397,-65.557,-177.578,7.552,148.730
C04534=1157.677,239.645,-65.584,-177.575,7.555,148.730
C04535=1157.673,239.893,-65.611,-177.573,7.557,148.730
C04536=1157.669,240.142,-65.637,-177.570,7.560,148.730
C04537=1157.664,240.391,-65.664,-177.567,7.563,148.730
C04538=1157.659,240.639,-65.691,-177.564,7.565,148.730
C04539=1157.655,240.887,-65.717,-177.562,7.567,148.730
C04540=1157.650,241.136,-65.744,-177.559,7.570,148.729
C04541=1157.646,241.385,-65.770,-177.556,7.573,148.729
C04542=1157.642,241.633,-65.797,-177.553,7.576,148.729
C04543=1157.637,241.882,-65.824,-177.551,7.579,148.729
C04544=1157.633,242.130,-65.851,-177.548,7.581,148.729
C04545=1157.628,242.379,-65.877,-177.545,7.584,148.729
C04546=1157.624,242.627,-65.904,-177.542,7.587,148.729
C04547=1157.620,242.875,-65.930,-177.540,7.590,148.729
C04548=1157.615,243.124,-65.958,-177.537,7.593,148.729
C04549=1157.610,243.372,-65.985,-177.535,7.595,148.729
C04550=1157.606,243.621,-66.011,-177.532,7.598,148.728
C04551=1157.602,243.869,-66.038,-177.529,7.600,148.728
C04552=1157.597,244.118,-66.065,-177.526,7.603,148.728
C04553=1157.592,244.366,-66.092,-177.523,7.606,148.728
C04554=1157.589,244.615,-66.119,-177.521,7.608,148.728
C04555=1157.585,244.864,-66.146,-177.518,7.611,148.728
C04556=1157.580,245.112,-66.173,-177.515,7.614,148.728
C04557=1157.575,245.361,-66.200,-177.512,7.617,148.728
C04558=1157.571,245.609,-66.227,-177.509,7.620,148.727
C04559=1157.567,245.857,-66.254,-177.507,7.622,148.727
C04560=1157.562,246.106,-66.281,-177.504,7.625,148.727
C04561=1157.557,246.354,-66.308,-177.502,7.628,148.727
C04562=1157.554,246.603,-66.335,-177.499,7.631,148.727
C04563=1157.549,246.852,-66.362,-177.496,7.634,148.727
C04564=1157.545,247.100,-66.389,-177.494,7.636,148.727
C04565=1157.540,247.349,-66.416,-177.491,7.639,148.727
C04566=1157.535,247.597,-66.443,-177.488,7.642,148.727
C04567=1157.531,247.846,-66.470,-177.485,7.644,148.727
C04568=1157.527,248.094,-66.497,-177.482,7.647,148.726
C04569=1157.523,248.343,-66.524,-177.479,7.650,148.726
C04570=1157.518,248.591,-66.552,-177.477,7.652,148.726
C04571=1157.514,248.839,-66.579,-177.474,7.655,148.726
C04572=1157.509,249.088,-66.606,-177.472,7.658,148.726
C04573=1157.504,249.336,-66.633,-177.469,7.661,148.726
C04574=1157.500,249.586,-66.660,-177.466,7.664,148.726
C04575=1157.496,249.833,-66.688,-177.463,7.667,148.726
C04576=1157.491,250.082,-66.715,-177.461,7.669,148.726
C04577=1157.487,250.330,-66.742,-177.458,7.672,148.726
C04578=1157.483,250.579,-66.769,-177.455,7.675,148.725
C04579=1157.479,250.827,-66.797,-177.452,7.677,148.725
C04580=1157.474,251.076,-66.824,-177.450,7.680,148.725
C04581=1157.470,251.324,-66.851,-177.447,7.683,148.725
C04582=1157.465,251.572,-66.879,-177.445,7.685,148.725
C04583=1157.461,251.821,-66.906,-177.442,7.688,148.725
C04584=1157.457,252.070,-66.933,-177.439,7.691,148.725
C04585=1157.452,252.318,-66.961,-177.436,7.694,148.725
C04586=1157.448,252.567,-66.988,-177.434,7.697,148.725
C04587=1157.444,252.815,-67.016,-177.431,7.700,148.725
C04588=1157.439,253.063,-67.043,-177.428,7.703,148.725
C04589=1157.435,253.312,-67.070,-177.426,7.705,148.725
C04590=1157.431,253.560,-67.098,-177.423,7.708,148.725
C04591=1157.426,253.809,-67.126,-177.420,7.711,148.725
C04592=1157.422,254.057,-67.153,-177.418,7.714,148.724
C04593=1157.417,254.306,-67.181,-177.415,7.717,148.724
C04594=1157.413,254.554,-67.209,-177.412,7.720,148.724
C04595=1157.408,254.802,-67.236,-177.409,7.723,148.724
C04596=1157.404,255.051,-67.264,-177.407,7.725,148.724
C04597=1157.400,255.300,-67.291,-177.404,7.728,148.724
C04598=1157.395,255.547,-67.319,-177.401,7.731,148.724
C04599=1157.391,255.797,-67.347,-177.398,7.734,148.724
C04600=1157.387,256.044,-67.374,-177.396,7.736,148.724
C04601=1157.382,256.293,-67.401,-177.393,7.739,148.724
C04602=1157.378,256.542,-67.430,-177.390,7.742,148.724
C04603=1157.373,256.790,-67.457,-177.387,7.745,148.724
C04604=1157.369,257.038,-67.485,-177.385,7.747,148.723
C04605=1157.365,257.287,-67.513,-177.382,7.750,148.723
C04606=1157.360,257.535,-67.540,-177.379,7.753,148.723
C04607=1157.356,257.783,-67.568,-177.377,7.756,148.723
C04608=1157.351,258.032,-67.597,-177.374,7.759,148.723
C04609=1157.347,258.281,-67.624,-177.371,7.762,148.723
C04610=1157.343,258.529,-67.652,-177.368,7.765,148.723
C04611=1157.339,258.777,-67.680,-177.366,7.768,148.723
C04612=1157.334,259.026,-67.707,-177.363,7.771,148.723
C04613=1157.330,259.274,-67.736,-177.360,7.774,148.723
C04614=1157.325,259.522,-67.763,-177.358,7.776,148.723
C04615=1157.321,259.771,-67.791,-177.356,7.779,148.723
C04616=1157.317,260.019,-67.818,-177.353,7.782,148.723
C04617=1157.312,260.268,-67.847,-177.350,7.785,148.723
C04618=1157.308,260.516,-67.875,-177.347,7.788,148.723
C04619=1157.304,260.764,-67.903,-177.345,7.791,148.723
C04620=1157.299,261.013,-67.932,-177.342,7.794,148.723
C04621=1157.295,261.261,-67.959,-177.339,7.797,148.723
C04622=1157.290,261.534,-67.990,-177.336,7.800,148.723
C04623=1157.285,261.807,-68.021,-177.333,7.803,148.722
C04624=1157.281,262.081,-68.051,-177.330,7.807,148.722
C04625=1157.275,262.354,-68.083,-177.327,7.810,148.722
C04626=1157.272,262.603,-68.111,-177.325,7.813,148.722
C04627=1157.267,262.851,-68.139,-177.322,7.816,148.722
C04628=1157.263,263.100,-68.167,-177.319,7.818,148.722
C04629=1157.258,263.348,-68.195,-177.316,7.821,148.722
C04630=1157.255,263.596,-68.223,-177.313,7.824,148.722
C04631=1157.250,263.844,-68.252,-177.311,7.827,148.722
C04632=1157.246,264.093,-68.280,-177.309,7.829,148.722
C04633=1157.241,264.341,-68.308,-177.306,7.832,148.722
C04634=1157.237,264.590,-68.336,-177.303,7.835,148.722
C04635=1157.232,264.838,-68.365,-177.300,7.838,148.722
C04636=1157.228,265.086,-68.393,-177.297,7.841,148.722
C04637=1157.224,265.334,-68.421,-177.295,7.844,148.722
C04638=1157.219,265.583,-68.449,-177.292,7.847,148.722
C04639=1157.215,265.831,-68.477,-177.290,7.850,148.722
C04640=1157.210,266.080,-68.506,-177.287,7.853,148.722
C04641=1157.206,266.328,-68.534,-177.284,7.856,148.722
C04642=1157.202,266.577,-68.562,-177.281,7.859,148.722
C04643=1157.198,266.825,-68.591,-177.279,7.862,148.722
C04644=1157.193,267.073,-68.620,-177.276,7.865,148.722
C04645=1157.189,267.321,-68.648,-177.273,7.868,148.721
C04646=1157.184,267.570,-68.676,-177.270,7.871,148.721
C04647=1157.180,267.819,-68.705,-177.267,7.874,148.721
C04648=1157.175,268.066,-68.733,-177.266,7.876,148.721
C04649=1157.171,268.315,-68.762,-177.263,7.879,148.721
C04650=1157.168,268.563,-68.790,-177.260,7.882,148.721
C04651=1157.162,268.811,-68.819,-177.257,7.885,148.721
C04652=1157.159,269.060,-68.847,-177.255,7.888,148.721
C04653=1157.154,269.308,-68.876,-177.252,7.891,148.721
C04654=1157.149,269.556,-68.904,-177.249,7.894,148.721
C04655=1157.146,269.805,-68.933,-177.246,7.897,148.721
C04656=1157.141,270.053,-68.962,-177.244,7.900,148.721
C04657=1157.137,270.301,-68.990,-177.241,7.903,148.721
C04658=1157.133,270.550,-69.019,-177.239,7.906,148.721
C04659=1157.128,270.798,-69.048,-177.236,7.909,148.721
C04660=1157.124,271.046,-69.076,-177.233,7.912,148.721
C04661=1157.120,271.295,-69.105,-177.230,7.915,148.721
C04662=1157.115,271.543,-69.134,-177.228,7.918,148.721
C04663=1157.111,271.791,-69.162,-177.225,7.921,148.721
C04664=1157.107,272.040,-69.191,-177.222,7.924,148.721
C04665=1157.102,272.288,-69.220,-177.220,7.927,148.721
C04666=1157.098,272.536,-69.248,-177.217,7.930,148.721
C04667=1157.094,272.785,-69.277,-177.214,7.933,148.721
C04668=1157.089,273.033,-69.306,-177.212,7.936,148.721
C04669=1157.085,273.281,-69.335,-177.209,7.939,148.721
C04670=1157.081,273.530,-69.363,-177.206,7.942,148.721
C04671=1157.077,273.778,-69.393,-177.204,7.945,148.721
C04672=1157.072,274.026,-69.421,-177.201,7.948,148.721
C04673=1157.067,274.274,-69.450,-177.198,7.951,148.721
C04674=1157.064,274.523,-69.479,-177.196,7.954,148.721
C04675=1157.059,274.771,-69.508,-177.193,7.957,148.721
C04676=1157.055,275.019,-69.537,-177.190,7.960,148.721
C04677=1157.050,275.268,-69.566,-177.187,7.963,148.721
C04678=1157.047,275.516,-69.595,-177.185,7.966,148.721
C04679=1157.042,275.764,-69.623,-177.182,7.969,148.721
C04680=1157.037,276.012,-69.653,-177.180,7.972,148.721
C04681=1157.033,276.260,-69.682,-177.177,7.975,148.721
C04682=1157.029,276.509,-69.711,-177.174,7.978,148.721
C04683=1157.025,276.757,-69.740,-177.172,7.982,148.721
C04684=1157.021,277.005,-69.769,-177.169,7.985,148.721
C04685=1157.016,277.254,-69.797,-177.166,7.988,148.721
C04686=1157.012,277.502,-69.827,-177.163,7.990,148.721
C04687=1157.008,277.750,-69.856,-177.161,7.993,148.721
C04688=1157.004,277.998,-69.886,-177.158,7.997,148.721
C04689=1156.999,278.247,-69.915,-177.156,8.000,148.721
C04690=1156.995,278.496,-69.944,-177.153,8.003,148.721
C04691=1156.990,278.743,-69.973,-177.150,8.006,148.721
C04692=1156.986,278.991,-70.003,-177.148,8.009,148.721
C04693=1156.982,279.239,-70.031,-177.145,8.012,148.721
C04694=1156.978,279.488,-70.060,-177.142,8.015,148.721
C04695=1156.974,279.736,-70.090,-177.139,8.018,148.721
C04696=1156.970,279.985,-70.119,-177.137,8.021,148.721
C04697=1156.965,280.232,-70.148,-177.134,8.024,148.721
C04698=1156.961,280.481,-70.178,-177.132,8.027,148.721
C04699=1156.956,280.729,-70.207,-177.129,8.030,148.721
C04700=1156.952,280.977,-70.236,-177.127,8.033,148.721
C04701=1156.948,281.225,-70.266,-177.124,8.036,148.721
C04702=1156.944,281.474,-70.295,-177.121,8.039,148.721
C04703=1156.939,281.723,-70.324,-177.119,8.042,148.721
C04704=1156.935,281.971,-70.354,-177.116,8.045,148.721
C04705=1156.930,282.218,-70.383,-177.113,8.048,148.721
C04706=1156.926,282.467,-70.412,-177.110,8.051,148.721
C04707=1156.921,282.715,-70.442,-177.108,8.054,148.721
C04708=1156.917,282.964,-70.472,-177.105,8.057,148.721
C04709=1156.913,283.212,-70.501,-177.103,8.060,148.721
C04710=1156.909,283.460,-70.531,-177.100,8.064,148.721
C04711=1156.905,283.708,-70.561,-177.097,8.067,148.721
C04712=1156.901,283.956,-70.590,-177.095,8.070,148.721
C04713=1156.897,284.204,-70.620,-177.092,8.074,148.721
C04714=1156.892,284.452,-70.649,-177.089,8.077,148.721
C04715=1156.888,284.701,-70.679,-177.086,8.080,148.721
C04716=1156.884,284.949,-70.708,-177.084,8.082,148.721
C04717=1156.879,285.198,-70.738,-177.081,8.086,148.721
C04718=1156.875,285.446,-70.767,-177.078,8.089,148.721
C04719=1156.871,285.694,-70.797,-177.076,8.092,148.721
C04720=1156.867,285.942,-70.827,-177.073,8.095,148.721
C04721=1156.863,286.190,-70.857,-177.071,8.098,148.721
C04722=1156.859,286.438,-70.886,-177.068,8.101,148.721
C04723=1156.854,286.687,-70.916,-177.066,8.104,148.722
C04724=1156.850,286.935,-70.946,-177.063,8.107,148.722
C04725=1156.846,287.183,-70.976,-177.060,8.110,148.721
C04726=1156.841,287.458,-71.008,-177.057,8.114,148.722
C04727=1156.836,287.733,-71.042,-177.054,8.117,148.722
C04728=1156.831,288.008,-71.074,-177.051,8.121,148.722
C04729=1156.826,288.283,-71.107,-177.049,8.124,148.722
C04730=1156.822,288.531,-71.137,-177.046,8.127,148.722
C04731=1156.818,288.779,-71.168,-177.043,8.130,148.722
C04732=1156.813,289.028,-71.197,-177.041,8.133,148.722
C04733=1156.809,289.276,-71.227,-177.038,8.137,148.722
C04734=1156.805,289.524,-71.257,-177.035,8.140,148.722
C04735=1156.800,289.772,-71.287,-177.033,8.143,148.722
C04736=1156.796,290.020,-71.316,-177.030,8.146,148.722
C04737=1156.792,290.269,-71.347,-177.027,8.150,148.722
C04738=1156.788,290.517,-71.377,-177.025,8.152,148.722
C04739=1156.784,290.765,-71.407,-177.022,8.155,148.722
C04740=1156.779,291.014,-71.437,-177.020,8.159,148.722
C04741=1156.775,291.261,-71.467,-177.017,8.162,148.722
C04742=1156.771,291.509,-71.497,-177.015,8.165,148.722
C04743=1156.767,291.757,-71.527,-177.012,8.168,148.722
C04744=1156.762,292.006,-71.557,-177.008,8.172,148.722
C04745=1156.759,292.253,-71.587,-177.006,8.175,148.723
C04746=1156.754,292.503,-71.618,-177.003,8.178,148.723
C04747=1156.750,292.750,-71.648,-177.001,8.181,148.723
C04748=1156.745,292.999,-71.678,-176.998,8.184,148.723
C04749=1156.742,293.246,-71.708,-176.996,8.187,148.723
C04750=1156.738,293.494,-71.738,-176.993,8.190,148.723
C04751=1156.733,293.743,-71.768,-176.990,8.193,148.723
C04752=1156.729,293.990,-71.798,-176.988,8.197,148.723
C04753=1156.725,294.240,-71.829,-176.985,8.200,148.723
C04754=1156.721,294.487,-71.859,-176.983,8.204,148.723
C04755=1156.716,294.735,-71.890,-176.980,8.207,148.723
C04756=1156.712,294.983,-71.919,-176.977,8.210,148.723
C04757=1156.707,295.231,-71.950,-176.975,8.213,148.723
C04758=1156.703,295.479,-71.980,-176.972,8.216,148.723
C04759=1156.699,295.728,-72.011,-176.970,8.219,148.723
C04760=1156.695,295.976,-72.041,-176.967,8.222,148.723
C04761=1156.691,296.224,-72.071,-176.965,8.225,148.724
C04762=1156.687,296.472,-72.102,-176.962,8.228,148.724
C04763=1156.683,296.720,-72.133,-176.959,8.232,148.724
C04764=1156.679,296.969,-72.162,-176.956,8.235,148.724
C04765=1156.674,297.216,-72.193,-176.954,8.239,148.724
C04766=1156.669,297.464,-72.224,-176.951,8.242,148.724
C04767=1156.665,297.712,-72.254,-176.949,8.245,148.724
C04768=1156.661,297.961,-72.285,-176.946,8.248,148.724
C04769=1156.657,298.209,-72.314,-176.944,8.251,148.724
C04770=1156.653,298.457,-72.345,-176.941,8.254,148.724
C04771=1156.648,298.705,-72.376,-176.938,8.258,148.724
C04772=1156.645,298.953,-72.406,-176.935,8.261,148.724
C04773=1156.640,299.201,-72.437,-176.933,8.264,148.724
C04774=1156.636,299.449,-72.468,-176.930,8.267,148.724
C04775=1156.632,299.697,-72.498,-176.928,8.271,148.725
C04776=1156.628,299.946,-72.529,-176.925,8.274,148.725
C04777=1156.623,300.193,-72.560,-176.923,8.277,148.725
C04778=1156.619,300.441,-72.590,-176.920,8.281,148.725
C04779=1156.615,300.690,-72.621,-176.917,8.284,148.725
C04780=1156.611,300.938,-72.652,-176.914,8.287,148.725
C04781=1156.607,301.185,-72.682,-176.912,8.290,148.725
C04782=1156.603,301.434,-72.713,-176.909,8.293,148.725
C04783=1156.598,301.682,-72.744,-176.907,8.296,148.725
C04784=1156.594,301.930,-72.774,-176.904,8.299,148.725
C04785=1156.590,302.178,-72.805,-176.901,8.303,148.725
C04786=1156.586,302.426,-72.836,-176.899,8.306,148.725
C04787=1156.581,302.674,-72.867,-176.896,8.310,148.726
C04788=1156.577,302.923,-72.898,-176.894,8.313,148.726
C04789=1156.573,303.171,-72.928,-176.891,8.316,148.726
C04790=1156.569,303.418,-72.960,-176.889,8.319,148.726
C04791=1156.565,303.667,-72.991,-176.886,8.322,148.726
C04792=1156.560,303.914,-73.022,-176.883,8.326,148.726
C04793=1156.555,304.162,-73.052,-176.881,8.329,148.726
C04794=1156.552,304.411,-73.083,-176.878,8.332,148.726
C04795=1156.548,304.658,-73.114,-176.876,8.335,148.726
C04796=1156.543,304.906,-73.145,-176.873,8.339,148.726
C04797=1156.539,305.155,-73.176,-176.870,8.342,148.726
C04798=1156.535,305.403,-73.207,-176.868,8.346,148.727
C04799=1156.531,305.651,-73.239,-176.865,8.349,148.727
C04800=1156.526,305.899,-73.270,-176.862,8.352,148.727
C04801=1156.522,306.147,-73.300,-176.860,8.355,148.727
C04802=1156.518,306.395,-73.331,-176.857,8.358,148.727
C04803=1156.514,306.642,-73.363,-176.855,8.362,148.727
C04804=1156.510,306.891,-73.394,-176.852,8.366,148.727
C04805=1156.506,307.139,-73.424,-176.849,8.369,148.727
C04806=1156.502,307.387,-73.456,-176.847,8.372,148.728
C04807=1156.497,307.635,-73.487,-176.844,8.375,148.728
C04808=1156.493,307.882,-73.518,-176.842,8.378,148.728
C04809=1156.489,308.131,-73.550,-176.839,8.382,148.728
C04810=1156.484,308.379,-73.580,-176.836,8.385,148.728
C04811=1156.481,308.627,-73.612,-176.834,8.388,148.728
C04812=1156.476,308.875,-73.643,-176.831,8.391,148.728
C04813=1156.472,309.123,-73.675,-176.829,8.395,148.728
C04814=1156.468,309.371,-73.706,-176.826,8.399,148.728
C04815=1156.464,309.619,-73.737,-176.823,8.402,148.728
C04816=1156.459,309.867,-73.768,-176.821,8.405,148.729
C04817=1156.456,310.115,-73.800,-176.819,8.408,148.729
C04818=1156.451,310.363,-73.831,-176.816,8.411,148.729
C04819=1156.447,310.611,-73.863,-176.813,8.415,148.729
C04820=1156.443,310.859,-73.893,-176.810,8.418,148.729
C04821=1156.439,311.107,-73.925,-176.808,8.422,148.729
C04822=1156.435,311.354,-73.957,-176.806,8.425,148.729
C04823=1156.431,311.603,-73.988,-176.803,8.428,148.729
C04824=1156.426,311.850,-74.019,-176.800,8.432,148.730
C04825=1156.422,312.099,-74.051,-176.798,8.435,148.730
C04826=1156.417,312.347,-74.083,-176.795,8.438,148.730
C04827=1156.414,312.595,-74.114,-176.793,8.441,148.730
C04828=1156.410,312.843,-74.146,-176.790,8.445,148.730
C04829=1156.405,313.091,-74.177,-176.787,8.449,148.730
C04830=1156.401,313.368,-74.213,-176.785,8.452,148.730
C04831=1156.396,313.645,-74.248,-176.782,8.456,148.731
C04832=1156.391,313.923,-74.283,-176.779,8.460,148.731
C04833=1156.387,314.201,-74.318,-176.776,8.464,148.731
C04834=1156.383,314.448,-74.350,-176.773,8.467,148.731
C04835=1156.378,314.696,-74.382,-176.771,8.470,148.731
C04836=1156.374,314.944,-74.414,-176.768,8.473,148.731
C04837=1156.370,315.192,-74.445,-176.766,8.477,148.731
C04838=1156.366,315.440,-74.477,-176.763,8.481,148.732
C04839=1156.362,315.688,-74.508,-176.760,8.484,148.732
C04840=1156.358,315.936,-74.541,-176.758,8.487,148.732
C04841=1156.353,316.183,-74.572,-176.756,8.490,148.732
C04842=1156.350,316.431,-74.604,-176.752,8.494,148.732
C04843=1156.346,316.679,-74.636,-176.750,8.497,148.732
C04844=1156.340,316.928,-74.667,-176.748,8.501,148.732
C04845=1156.337,317.176,-74.699,-176.745,8.504,148.733
C04846=1156.333,317.424,-74.731,-176.742,8.508,148.733
C04847=1156.329,317.671,-74.762,-176.740,8.511,148.733
C04848=1156.324,317.919,-74.795,-176.738,8.514,148.733
C04849=1156.321,318.168,-74.827,-176.735,8.517,148.733
C04850=1156.316,318.415,-74.858,-176.732,8.521,148.733
C04851=1156.312,318.663,-74.891,-176.730,8.524,148.733
C04852=1156.308,318.911,-74.922,-176.727,8.528,148.734
C04853=1156.304,319.159,-74.954,-176.725,8.531,148.734
C04854=1156.299,319.407,-74.986,-176.722,8.535,148.734
C04855=1156.296,319.655,-75.018,-176.719,8.538,148.734
C04856=1156.292,319.903,-75.050,-176.717,8.541,148.734
C04857=1156.287,320.150,-75.083,-176.715,8.545,148.734
C04858=1156.284,320.398,-75.115,-176.711,8.548,148.734
C04859=1156.279,320.646,-75.147,-176.709,8.552,148.735
C04860=1156.275,320.894,-75.179,-176.707,8.555,148.735
C04861=1156.271,321.142,-75.210,-176.704,8.558,148.735
C04862=1156.267,321.390,-75.243,-176.702,8.562,148.735
C04863=1156.263,321.638,-75.275,-176.699,8.565,148.735
C04864=1156.259,321.886,-75.308,-176.696,8.569,148.735
C04865=1156.254,322.133,-75.339,-176.694,8.573,148.736
C04866=1156.251,322.381,-75.371,-176.691,8.576,148.736
C04867=1156.246,322.630,-75.404,-176.689,8.579,148.736
C04868=1156.243,322.878,-75.435,-176.686,8.582,148.736
C04869=1156.238,323.125,-75.469,-176.683,8.586,148.736
C04870=1156.234,323.373,-75.500,-176.681,8.590,148.736
C04871=1156.230,323.621,-75.533,-176.679,8.593,148.737
C04872=1156.226,323.869,-75.565,-176.676,8.596,148.737
C04873=1156.222,324.117,-75.598,-176.673,8.600,148.737
C04874=1156.218,324.365,-75.629,-176.671,8.603,148.737
C04875=1156.213,324.612,-75.662,-176.668,8.607,148.737
C04876=1156.210,324.860,-75.694,-176.666,8.611,148.737
C04877=1156.205,325.108,-75.726,-176.663,8.614,148.738
C04878=1156.201,325.356,-75.760,-176.661,8.617,148.738
C04879=1156.197,325.604,-75.791,-176.658,8.621,148.738
C04880=1156.193,325.852,-75.824,-176.655,8.624,148.738
C04881=1156.189,326.099,-75.856,-176.653,8.628,148.738
C04882=1156.185,326.348,-75.889,-176.651,8.631,148.738
C04883=1156.180,326.595,-75.922,-176.648,8.635,148.739
C04884=1156.177,326.843,-75.954,-176.645,8.638,148.739
C04885=1156.173,327.091,-75.987,-176.643,8.641,148.739
C04886=1156.169,327.339,-76.019,-176.640,8.646,148.739
C04887=1156.165,327.587,-76.052,-176.638,8.649,148.739
C04888=1156.160,327.835,-76.084,-176.635,8.652,148.740
C04889=1156.156,328.082,-76.116,-176.632,8.656,148.740
C04890=1156.152,328.330,-76.149,-176.630,8.659,148.740
C04891=1156.148,328.578,-76.182,-176.628,8.662,148.740
C04892=1156.144,328.826,-76.214,-176.625,8.666,148.740
C04893=1156.140,329.074,-76.247,-176.623,8.670,148.741
C04894=1156.136,329.321,-76.280,-176.620,8.673,148.741
C04895=1156.131,329.570,-76.313,-176.618,8.676,148.741
C04896=1156.128,329.817,-76.345,-176.615,8.680,148.741
C04897=1156.124,330.065,-76.378,-176.612,8.683,148.741
C04898=1156.119,330.313,-76.411,-176.610,8.687,148.741
C04899=1156.115,330.561,-76.444,-176.607,8.691,148.742
C04900=1156.112,330.808,-76.476,-176.605,8.694,148.742
C04901=1156.107,331.056,-76.508,-176.602,8.697,148.742
C04902=1156.103,331.304,-76.542,-176.600,8.702,148.742
C04903=1156.098,331.552,-76.575,-176.597,8.705,148.743
C04904=1156.095,331.800,-76.607,-176.595,8.708,148.743
C04905=1156.091,332.047,-76.640,-176.592,8.712,148.743
C04906=1156.086,332.295,-76.673,-176.590,8.715,148.743
C04907=1156.082,332.543,-76.706,-176.587,8.719,148.743
C04908=1156.078,332.790,-76.739,-176.584,8.723,148.744
C04909=1156.074,333.039,-76.772,-176.582,8.726,148.744
C04910=1156.070,333.286,-76.804,-176.580,8.729,148.744
C04911=1156.066,333.534,-76.837,-176.577,8.733,148.744
C04912=1156.062,333.782,-76.871,-176.574,8.736,148.744
C04913=1156.058,334.029,-76.904,-176.572,8.740,148.744
C04914=1156.054,334.277,-76.937,-176.569,8.744,148.745
C04915=1156.050,334.525,-76.970,-176.567,8.747,148.745
C04916=1156.046,334.773,-77.003,-176.564,8.751,148.745
C04917=1156.041,335.020,-77.036,-176.562,8.754,148.745
C04918=1156.038,335.269,-77.069,-176.559,8.758,148.746
C04919=1156.034,335.517,-77.102,-176.556,8.762,148.746
C04920=1156.030,335.765,-77.135,-176.554,8.765,148.746
C04921=1156.026,336.012,-77.168,-176.552,8.768,148.746
C04922=1156.022,336.260,-77.201,-176.549,8.773,148.746
C04923=1156.018,336.508,-77.234,-176.546,8.776,148.747
C04924=1156.013,336.755,-77.267,-176.544,8.779,148.747
C04925=1156.010,337.003,-77.301,-176.541,8.783,148.747
C04926=1156.005,337.250,-77.335,-176.539,8.786,148.747
C04927=1156.001,337.498,-77.368,-176.536,8.791,148.748
C04928=1155.997,337.746,-77.401,-176.534,8.794,148.748
C04929=1155.993,337.993,-77.434,-176.531,8.797,148.748
C04930=1155.990,338.242,-77.468,-176.529,8.801,148.748
C04931=1155.985,338.490,-77.501,-176.527,8.805,148.749
C04932=1155.981,338.737,-77.534,-176.524,8.808,148.749
C04933=1155.977,338.985,-77.567,-176.521,8.812,148.749
C04934=1155.972,339.265,-77.605,-176.519,8.816,148.749
C04935=1155.968,339.545,-77.643,-176.516,8.820,148.750
C04936=1155.963,339.825,-77.681,-176.513,8.824,148.750
C04937=1155.959,340.104,-77.718,-176.510,8.829,148.750
C04938=1155.954,340.352,-77.751,-176.508,8.832,148.750
C04939=1155.950,340.600,-77.786,-176.505,8.835,148.750
C04940=1155.946,340.848,-77.819,-176.502,8.839,148.751
C04941=1155.942,341.096,-77.852,-176.500,8.843,148.751
C04942=1155.938,341.344,-77.886,-176.497,8.847,148.751
C04943=1155.934,341.591,-77.919,-176.495,8.850,148.751
C04944=1155.930,341.838,-77.953,-176.492,8.854,148.752
C04945=1155.926,342.087,-77.987,-176.490,8.857,148.752
C04946=1155.922,342.334,-78.021,-176.488,8.861,148.752
C04947=1155.918,342.582,-78.054,-176.485,8.865,148.753
C04948=1155.914,342.829,-78.088,-176.483,8.868,148.753
C04949=1155.910,343.077,-78.121,-176.480,8.872,148.753
C04950=1155.906,343.326,-78.155,-176.477,8.876,148.753
C04951=1155.902,343.573,-78.189,-176.475,8.879,148.753
C04952=1155.898,343.820,-78.222,-176.472,8.883,148.754
C04953=1155.894,344.067,-78.256,-176.470,8.886,148.754
C04954=1155.889,344.316,-78.289,-176.467,8.890,148.754
C04955=1155.886,344.563,-78.324,-176.465,8.894,148.754
C04956=1155.882,344.811,-78.357,-176.462,8.898,148.755
C04957=1155.878,345.058,-78.391,-176.460,8.901,148.755
C04958=1155.873,345.306,-78.424,-176.458,8.905,148.755
C04959=1155.870,345.554,-78.459,-176.455,8.909,148.755
C04960=1155.865,345.802,-78.492,-176.452,8.912,148.756
C04961=1155.861,346.049,-78.526,-176.450,8.916,148.756
C04962=1155.857,346.298,-78.560,-176.447,8.919,148.756
C04963=1155.854,346.545,-78.594,-176.445,8.924,148.757
C04964=1155.849,346.792,-78.628,-176.442,8.927,148.757
C04965=1155.845,347.040,-78.661,-176.440,8.930,148.757
C04966=1155.842,347.288,-78.696,-176.437,8.934,148.757
C04967=1155.837,347.535,-78.730,-176.435,8.938,148.757
C04968=1155.833,347.783,-78.763,-176.432,8.942,148.758
C04969=1155.830,348.031,-78.797,-176.430,8.945,148.758
C04970=1155.825,348.278,-78.832,-176.427,8.950,148.758
C04971=1155.821,348.526,-78.865,-176.425,8.953,148.759
C04972=1155.817,348.774,-78.900,-176.422,8.957,148.759
C04973=1155.813,349.021,-78.934,-176.420,8.960,148.759
C04974=1155.809,349.269,-78.967,-176.417,8.965,148.759
C04975=1155.805,349.517,-79.002,-176.415,8.968,148.760
C04976=1155.801,349.764,-79.036,-176.413,8.971,148.760
C04977=1155.797,350.011,-79.070,-176.410,8.975,148.760
C04978=1155.793,350.259,-79.104,-176.407,8.979,148.760
C04979=1155.789,350.507,-79.139,-176.405,8.983,148.761
C04980=1155.785,350.755,-79.172,-176.403,8.986,148.761
C04981=1155.781,351.002,-79.207,-176.400,8.990,148.761
C04982=1155.777,351.250,-79.241,-176.397,8.994,148.762
C04983=1155.773,351.498,-79.276,-176.395,8.998,148.762
C04984=1155.769,351.745,-79.309,-176.393,9.001,148.762
C04985=1155.765,351.993,-79.344,-176.390,9.005,148.762
C04986=1155.761,352.240,-79.378,-176.387,9.009,148.763
C04987=1155.757,352.487,-79.413,-176.385,9.013,148.763
C04988=1155.753,352.735,-79.447,-176.383,9.016,148.763
C04989=1155.749,352.983,-79.481,-176.380,9.020,148.764
C04990=1155.745,353.231,-79.516,-176.378,9.024,148.764
C04991=1155.741,353.478,-79.550,-176.375,9.028,148.764
C04992=1155.737,353.726,-79.585,-176.373,9.031,148.764
C04993=1155.733,353.973,-79.619,-176.370,9.036,148.765
C04994=1155.729,354.221,-79.653,-176.368,9.039,148.765
C04995=1155.726,354.468,-79.687,-176.365,9.043,148.765
C04996=1155.721,354.716,-79.722,-176.363,9.047,148.766
C04997=1155.717,354.964,-79.757,-176.360,9.051,148.766
C04998=1155.713,355.211,-79.791,-176.358,9.054,148.766
C04999=1155.709,355.459,-79.825,-176.355,9.058,148.767
C05000=1155.705,355.707,-79.860,-176.353,9.062,148.767
C05001=1155.701,355.954,-79.894,-176.350,9.066,148.767
C05002=1155.697,356.201,-79.929,-176.348,9.069,148.767
C05003=1155.693,356.449,-79.964,-176.345,9.073,148.768
C05004=1155.689,356.696,-79.998,-176.343,9.077,148.768
C05005=1155.685,356.945,-80.033,-176.340,9.081,148.768
C05006=1155.681,357.192,-80.067,-176.338,9.084,148.769
C05007=1155.678,357.439,-80.102,-176.335,9.088,148.769
C05008=1155.673,357.687,-80.137,-176.333,9.092,148.769
C05009=1155.669,357.935,-80.172,-176.330,9.096,148.770
C05010=1155.665,358.183,-80.206,-176.328,9.099,148.770
C05011=1155.662,358.429,-80.241,-176.326,9.104,148.770
C05012=1155.658,358.677,-80.276,-176.323,9.108,148.771
C05013=1155.653,358.925,-80.310,-176.320,9.111,148.771
C05014=1155.650,359.172,-80.346,-176.318,9.116,148.771
C05015=1155.646,359.419,-80.380,-176.316,9.119,148.771
C05016=1155.642,359.668,-80.414,-176.313,9.123,148.772
C05017=1155.638,359.915,-80.450,-176.311,9.127,148.772
C05018=1155.634,360.162,-80.484,-176.308,9.131,148.772
C05019=1155.630,360.410,-80.520,-176.305,9.135,148.773
C05020=1155.626,360.657,-80.554,-176.303,9.138,148.773
C05021=1155.622,360.905,-80.589,-176.300,9.142,148.773
C05022=1155.618,361.153,-80.624,-176.298,9.146,148.774
C05023=1155.614,361.399,-80.659,-176.295,9.150,148.774
C05024=1155.610,361.648,-80.694,-176.293,9.154,148.774
C05025=1155.607,361.895,-80.730,-176.290,9.158,148.774
C05026=1155.602,362.143,-80.764,-176.288,9.162,148.775
C05027=1155.598,362.390,-80.800,-176.285,9.166,148.775
C05028=1155.595,362.638,-80.834,-176.283,9.170,148.776
C05029=1155.591,362.885,-80.869,-176.280,9.174,148.776
C05030=1155.587,363.133,-80.904,-176.278,9.177,148.776
C05031=1155.583,363.380,-80.940,-176.275,9.181,148.777
C05032=1155.579,363.628,-80.974,-176.272,9.185,148.777
C05033=1155.575,363.875,-81.010,-176.271,9.189,148.777
C05034=1155.571,364.123,-81.045,-176.268,9.193,148.778
C05035=1155.567,364.370,-81.080,-176.265,9.198,148.778
C05036=1155.563,364.618,-81.115,-176.263,9.201,148.778
C05037=1155.559,364.865,-81.151,-176.260,9.205,148.779
C05038=1155.555,365.147,-81.191,-176.258,9.209,148.779
C05039=1155.551,365.431,-81.231,-176.255,9.214,148.779
C05040=1155.546,365.713,-81.272,-176.252,9.219,148.780
C05041=1155.541,365.996,-81.312,-176.249,9.223,148.780
C05042=1155.537,366.244,-81.346,-176.247,9.228,148.781
C05043=1155.534,366.491,-81.382,-176.244,9.231,148.781
C05044=1155.530,366.739,-81.418,-176.242,9.235,148.781
C05045=1155.526,366.986,-81.453,-176.239,9.239,148.782
C05046=1155.521,367.234,-81.489,-176.237,9.243,148.782
C05047=1155.517,367.482,-81.524,-176.235,9.247,148.783
C05048=1155.514,367.729,-81.559,-176.232,9.251,148.783
C05049=1155.510,367.976,-81.594,-176.230,9.255,148.783
C05050=1155.506,368.223,-81.630,-176.227,9.259,148.784
C05051=1155.502,368.471,-81.666,-176.225,9.263,148.784
C05052=1155.499,368.719,-81.701,-176.223,9.267,148.784
C05053=1155.495,368.966,-81.737,-176.221,9.271,148.785
C05054=1155.491,369.213,-81.772,-176.218,9.275,148.785
C05055=1155.486,369.461,-81.808,-176.216,9.279,148.786
C05056=1155.483,369.708,-81.844,-176.213,9.283,148.786
C05057=1155.479,369.956,-81.879,-176.211,9.287,148.786
C05058=1155.475,370.203,-81.915,-176.209,9.291,148.787
C05059=1155.471,370.450,-81.950,-176.207,9.295,148.787
C05060=1155.467,370.698,-81.986,-176.205,9.299,148.788
C05061=1155.463,370.945,-82.021,-176.202,9.303,148.788
C05062=1155.459,371.193,-82.057,-176.200,9.307,148.789
C05063=1155.456,371.440,-82.093,-176.198,9.311,148.789
C05064=1155.452,371.688,-82.128,-176.196,9.315,148.790
C05065=1155.447,371.935,-82.164,-176.194,9.319,148.790
C05066=1155.443,372.182,-82.199,-176.192,9.323,148.790
C05067=1155.440,372.430,-82.235,-176.189,9.327,148.791
C05068=1155.436,372.677,-82.271,-176.188,9.331,148.792
C05069=1155.432,372.925,-82.307,-176.185,9.335,148.792
C05070=1155.428,373.172,-82.343,-176.183,9.339,148.792
C05071=1155.425,373.420,-82.378,-176.181,9.343,148.793
C05072=1155.420,373.667,-82.415,-176.179,9.347,148.794
C05073=1155.416,373.914,-82.450,-176.177,9.352,148.794
C05074=1155.412,374.162,-82.485,-176.175,9.355,148.794
C05075=1155.409,374.409,-82.522,-176.174,9.359,148.795
C05076=1155.404,374.656,-82.558,-176.171,9.364,148.796
C05077=1155.401,374.904,-82.593,-176.170,9.367,148.796
C05078=1155.397,375.151,-82.629,-176.168,9.371,148.797
C05079=1155.393,375.399,-82.666,-176.166,9.376,148.797
C05080=1155.389,375.646,-82.701,-176.164,9.379,148.798
C05081=1155.385,375.894,-82.737,-176.162,9.383,148.798
C05082=1155.382,376.141,-82.774,-176.161,9.387,148.799
C05083=1155.378,376.388,-82.809,-176.159,9.392,148.799
C05084=1155.374,376.636,-82.845,-176.157,9.395,148.800
C05085=1155.370,376.882,-82.881,-176.156,9.399,148.801
C05086=1155.365,377.130,-82.917,-176.154,9.403,148.801
C05087=1155.362,377.377,-82.954,-176.152,9.407,148.802
C05088=1155.358,377.624,-82.989,-176.151,9.411,148.802
C05089=1155.354,377.872,-83.025,-176.149,9.415,148.803
C05090=1155.350,378.119,-83.062,-176.147,9.419,148.804
C05091=1155.346,378.367,-83.098,-176.146,9.423,148.804
C05092=1155.343,378.614,-83.134,-176.144,9.427,148.805
C05093=1155.338,378.862,-83.170,-176.143,9.431,148.805
C05094=1155.335,379.108,-83.206,-176.141,9.435,148.806
C05095=1155.330,379.356,-83.243,-176.141,9.438,148.807
C05096=1155.327,379.603,-83.279,-176.140,9.442,148.807
C05097=1155.323,379.851,-83.315,-176.138,9.446,148.808
C05098=1155.319,380.098,-83.351,-176.137,9.450,148.809
C05099=1155.315,380.346,-83.387,-176.136,9.454,148.810
C05100=1155.312,380.593,-83.424,-176.134,9.458,148.810
C05101=1155.307,380.840,-83.460,-176.134,9.461,148.811
C05102=1155.304,381.087,-83.496,-176.132,9.465,148.812
C05103=1155.299,381.335,-83.532,-176.131,9.470,148.812
C05104=1155.296,381.582,-83.568,-176.130,9.473,148.813
C05105=1155.292,381.830,-83.605,-176.129,9.477,148.814
C05106=1155.288,382.077,-83.641,-176.128,9.481,148.814
C05107=1155.284,382.324,-83.678,-176.127,9.484,148.815
C05108=1155.281,382.571,-83.713,-176.126,9.488,148.816
C05109=1155.276,382.818,-83.750,-176.125,9.491,148.817
C05110=1155.272,383.066,-83.787,-176.125,9.495,148.817
C05111=1155.269,383.313,-83.823,-176.124,9.499,148.818
C05112=1155.265,383.561,-83.860,-176.123,9.502,148.819
C05113=1155.262,383.808,-83.896,-176.123,9.506,148.820
C05114=1155.257,384.056,-83.932,-176.122,9.510,148.820
C05115=1155.254,384.303,-83.968,-176.121,9.513,148.821
C05116=1155.250,384.550,-84.005,-176.121,9.517,148.822
C05117=1155.246,384.798,-84.041,-176.121,9.520,148.823
C05118=1155.242,385.045,-84.078,-176.120,9.524,148.823
C05119=1155.238,385.292,-84.115,-176.120,9.527,148.824
C05120=1155.235,385.539,-84.150,-176.119,9.530,148.825
C05121=1155.230,385.786,-84.187,-176.119,9.534,148.826
C05122=1155.226,386.034,-84.224,-176.119,9.537,148.827
C05123=1155.223,386.280,-84.260,-176.119,9.540,148.827
C05124=1155.219,386.528,-84.296,-176.119,9.544,148.828
C05125=1155.215,386.776,-84.333,-176.118,9.547,148.829
C05126=1155.212,387.023,-84.370,-176.118,9.550,148.830
C05127=1155.208,387.270,-84.407,-176.118,9.553,148.831
C05128=1155.203,387.518,-84.443,-176.119,9.556,148.832
C05129=1155.200,387.765,-84.479,-176.118,9.560,148.832
C05130=1155.196,388.012,-84.516,-176.119,9.562,148.833
C05131=1155.192,388.259,-84.552,-176.119,9.566,148.834
C05132=1155.188,388.506,-84.589,-176.119,9.568,148.835
C05133=1155.184,388.754,-84.625,-176.119,9.571,148.836
C05134=1155.181,389.001,-84.661,-176.119,9.575,148.837
C05135=1155.177,389.249,-84.699,-176.119,9.577,148.837
C05136=1155.173,389.496,-84.735,-176.119,9.580,148.838
C05137=1155.170,389.743,-84.772,-176.120,9.583,148.839
C05138=1155.165,389.991,-84.808,-176.121,9.586,148.840
C05139=1155.161,390.238,-84.845,-176.120,9.589,148.841
C05140=1155.158,390.485,-84.881,-176.121,9.592,148.842
C05141=1155.154,390.732,-84.918,-176.121,9.595,148.842
C05142=1155.149,391.019,-84.960,-176.122,9.598,148.843
C05143=1155.145,391.304,-85.003,-176.122,9.601,148.844
C05144=1155.140,391.591,-85.045,-176.123,9.604,148.845
C05145=1155.136,391.876,-85.087,-176.123,9.608,148.846
C05146=1155.132,392.124,-85.124,-176.124,9.610,148.847
C05147=1155.128,392.371,-85.160,-176.124,9.612,148.848
C05148=1155.125,392.619,-85.197,-176.125,9.615,148.849
C05149=1155.121,392.866,-85.234,-176.125,9.618,148.850
C05150=1155.117,393.113,-85.271,-176.126,9.620,148.850
C05151=1155.113,393.360,-85.308,-176.127,9.623,148.851
C05152=1155.109,393.607,-85.344,-176.127,9.625,148.852
C05153=1155.105,393.855,-85.380,-176.128,9.627,148.853
C05154=1155.101,394.102,-85.417,-176.129,9.630,148.854
C05155=1155.098,394.350,-85.453,-176.129,9.633,148.855
C05156=1155.094,394.597,-85.490,-176.130,9.635,148.855
C05157=1155.090,394.844,-85.527,-176.131,9.638,148.856
C05158=1155.086,395.091,-85.564,-176.131,9.640,148.857
C05159=1155.082,395.338,-85.600,-176.132,9.642,148.858
C05160=1155.078,395.585,-85.637,-176.133,9.645,148.859
C05161=1155.074,395.832,-85.674,-176.134,9.647,148.860
C05162=1155.071,396.080,-85.710,-176.134,9.649,148.860
C05163=1155.067,396.328,-85.747,-176.135,9.651,148.861
C05164=1155.063,396.575,-85.784,-176.136,9.654,148.862
C05165=1155.059,396.822,-85.821,-176.137,9.656,148.863
C05166=1155.056,397.069,-85.857,-176.138,9.658,148.864
C05167=1155.051,397.316,-85.894,-176.138,9.661,148.864
C05168=1155.047,397.563,-85.930,-176.139,9.663,148.865
C05169=1155.043,397.811,-85.967,-176.140,9.665,148.866
C05170=1155.040,398.058,-86.004,-176.141,9.667,148.867
C05171=1155.036,398.305,-86.041,-176.142,9.670,148.868
C05172=1155.032,398.553,-86.077,-176.142,9.671,148.868
C05173=1155.028,398.800,-86.114,-176.144,9.673,148.869
C05174=1155.025,399.047,-86.150,-176.144,9.676,148.870
C05175=1155.020,399.295,-86.187,-176.145,9.678,148.871
C05176=1155.016,399.542,-86.224,-176.146,9.680,148.872
C05177=1155.012,399.789,-86.261,-176.147,9.682,148.872
C05178=1155.010,400.036,-86.297,-176.148,9.684,148.873
C05179=1155.005,400.284,-86.334,-176.149,9.686,148.874
C05180=1155.001,400.531,-86.371,-176.149,9.688,148.875
C05181=1154.998,400.778,-86.407,-176.150,9.690,148.875
C05182=1154.994,401.025,-86.444,-176.151,9.692,148.876
C05183=1154.990,401.272,-86.481,-176.152,9.694,148.877
C05184=1154.986,401.521,-86.518,-176.153,9.696,148.878
C05185=1154.983,401.768,-86.554,-176.154,9.698,148.878
C05186=1154.979,402.015,-86.591,-176.154,9.700,148.879
C05187=1154.974,402.262,-86.627,-176.156,9.702,148.880
C05188=1154.970,402.509,-86.664,-176.156,9.704,148.880
C05189=1154.967,402.756,-86.701,-176.157,9.706,148.881
C05190=1154.963,403.003,-86.737,-176.158,9.707,148.882
C05191=1154.959,403.251,-86.775,-176.159,9.710,148.883
C05192=1154.955,403.498,-86.812,-176.159,9.712,148.884
C05193=1154.952,403.745,-86.848,-176.160,9.714,148.884
C05194=1154.948,403.992,-86.885,-176.161,9.716,148.885
C05195=1154.944,404.240,-86.922,-176.162,9.718,148.886
C05196=1154.940,404.487,-86.958,-176.163,9.720,148.886
C05197=1154.936,404.734,-86.994,-176.164,9.721,148.887
C05198=1154.933,404.982,-87.031,-176.165,9.724,148.888
C05199=1154.928,405.229,-87.068,-176.165,9.725,148.889
C05200=1154.924,405.476,-87.105,-176.166,9.727,148.889
C05201=1154.921,405.723,-87.141,-176.167,9.729,148.890
C05202=1154.917,405.971,-87.178,-176.168,9.731,148.891
C05203=1154.913,406.218,-87.215,-176.169,9.733,148.891
C05204=1154.909,406.465,-87.252,-176.169,9.734,148.892
C05205=1154.906,406.713,-87.288,-176.170,9.736,148.893
C05206=1154.902,406.960,-87.325,-176.171,9.738,148.894
C05207=1154.898,407.207,-87.362,-176.172,9.740,148.894
C05208=1154.894,407.454,-87.399,-176.172,9.742,148.895
C05209=1154.890,407.701,-87.436,-176.174,9.744,148.896
C05210=1154.886,407.948,-87.472,-176.174,9.745,148.896
C05211=1154.883,408.196,-87.509,-176.175,9.747,148.897
C05212=1154.879,408.443,-87.546,-176.176,9.749,148.898
C05213=1154.875,408.690,-87.583,-176.176,9.751,148.898
C05214=1154.871,408.937,-87.619,-176.177,9.753,148.899
C05215=1154.867,409.185,-87.655,-176.178,9.755,148.900
C05216=1154.863,409.432,-87.692,-176.179,9.756,148.900
C05217=1154.859,409.679,-87.729,-176.179,9.758,148.901
C05218=1154.856,409.927,-87.766,-176.180,9.760,148.902
C05219=1154.852,410.174,-87.803,-176.181,9.762,148.902
C05220=1154.848,410.421,-87.839,-176.181,9.763,148.903
C05221=1154.844,410.669,-87.876,-176.182,9.765,148.904
C05222=1154.840,410.916,-87.913,-176.183,9.767,148.904
C05223=1154.836,411.163,-87.949,-176.184,9.769,148.905
C05224=1154.833,411.411,-87.987,-176.184,9.770,148.905
C05225=1154.828,411.658,-88.024,-176.185,9.772,148.906
C05226=1154.824,411.905,-88.060,-176.185,9.775,148.907
C05227=1154.821,412.152,-88.097,-176.186,9.777,148.908
C05228=1154.817,412.399,-88.133,-176.187,9.778,148.908
C05229=1154.813,412.646,-88.170,-176.188,9.780,148.909
C05230=1154.809,412.894,-88.208,-176.188,9.782,148.910
C05231=1154.806,413.141,-88.244,-176.189,9.784,148.910
C05232=1154.802,413.388,-88.281,-176.189,9.785,148.911
C05233=1154.798,413.635,-88.318,-176.190,9.787,148.911
C05234=1154.794,413.883,-88.354,-176.191,9.789,148.912
C05235=1154.790,414.130,-88.391,-176.191,9.790,148.913
C05236=1154.786,414.377,-88.428,-176.191,9.793,148.913
C05237=1154.783,414.625,-88.465,-176.192,9.795,148.914
C05238=1154.779,414.872,-88.502,-176.193,9.796,148.915
C05239=1154.775,415.119,-88.538,-176.193,9.798,148.915
C05240=1154.773,415.366,-88.575,-176.194,9.800,148.916
C05241=1154.771,415.614,-88.611,-176.195,9.802,148.917
C05242=1154.770,416.020,-88.671,-176.195,9.805,148.917
C05243=1154.771,416.425,-88.730,-176.196,9.808,148.919
C05244=1154.774,416.830,-88.790,-176.197,9.811,148.919
C05245=1154.779,417.236,-88.848,-176.198,9.813,148.920
C05246=1154.358,417.237,-88.896,-176.200,9.824,148.924
C05247=1154.353,416.829,-88.837,-176.199,9.821,148.923
C05248=1154.350,416.421,-88.778,-176.199,9.818,148.922
C05249=1154.349,416.012,-88.718,-176.198,9.815,148.921
C05250=1154.350,415.602,-88.657,-176.197,9.812,148.920
C05251=1154.352,415.355,-88.621,-176.197,9.811,148.919
C05252=1154.354,415.108,-88.584,-176.196,9.809,148.919
C05253=1154.357,414.860,-88.547,-176.195,9.807,148.918
C05254=1154.361,414.613,-88.510,-176.195,9.805,148.917
C05255=1154.365,414.366,-88.473,-176.194,9.804,148.917
C05256=1154.369,414.119,-88.436,-176.193,9.802,148.916
C05257=1154.374,413.872,-88.400,-176.193,9.799,148.916
C05258=1154.377,413.625,-88.363,-176.192,9.798,148.915
C05259=1154.380,413.377,-88.326,-176.192,9.796,148.914
C05260=1154.384,413.130,-88.289,-176.192,9.794,148.914
C05261=1154.389,412.882,-88.252,-176.191,9.793,148.913
C05262=1154.393,412.635,-88.216,-176.190,9.791,148.912
C05263=1154.396,412.388,-88.179,-176.189,9.789,148.912
C05264=1154.400,412.141,-88.142,-176.188,9.787,148.911
C05265=1154.404,411.893,-88.105,-176.188,9.785,148.910
C05266=1154.408,411.646,-88.068,-176.187,9.784,148.910
C05267=1154.411,411.399,-88.032,-176.186,9.782,148.909
C05268=1154.415,411.151,-87.996,-176.186,9.780,148.908
C05269=1154.420,410.904,-87.959,-176.185,9.778,148.908
C05270=1154.424,410.657,-87.922,-176.185,9.776,148.907
C05271=1154.427,410.409,-87.885,-176.184,9.774,148.906
C05272=1154.431,410.162,-87.849,-176.183,9.772,148.906
C05273=1154.435,409.915,-87.812,-176.183,9.770,148.905
C05274=1154.439,409.668,-87.775,-176.182,9.769,148.905
C05275=1154.443,409.421,-87.738,-176.181,9.767,148.904
C05276=1154.446,409.174,-87.702,-176.180,9.765,148.903
C05277=1154.450,408.927,-87.665,-176.180,9.763,148.902
C05278=1154.454,408.679,-87.628,-176.179,9.761,148.902
C05279=1154.458,408.431,-87.591,-176.178,9.760,148.901
C05280=1154.461,408.185,-87.555,-176.178,9.758,148.900
C05281=1154.465,407.937,-87.518,-176.176,9.756,148.900
C05282=1154.469,407.690,-87.481,-176.176,9.754,148.899
C05283=1154.473,407.443,-87.444,-176.175,9.752,148.898
C05284=1154.477,407.195,-87.407,-176.174,9.751,148.898
C05285=1154.480,406.948,-87.371,-176.173,9.749,148.897
C05286=1154.484,406.701,-87.334,-176.173,9.747,148.896
C05287=1154.489,406.454,-87.297,-176.172,9.745,148.896
C05288=1154.493,406.207,-87.260,-176.171,9.743,148.895
C05289=1154.496,405.960,-87.224,-176.170,9.741,148.894
C05290=1154.499,405.712,-87.187,-176.169,9.739,148.893
C05291=1154.504,405.465,-87.150,-176.169,9.738,148.893
C05292=1154.508,405.218,-87.113,-176.168,9.736,148.892
C05293=1154.511,404.970,-87.077,-176.167,9.734,148.891
C05294=1154.515,404.723,-87.040,-176.166,9.732,148.891
C05295=1154.519,404.476,-87.004,-176.165,9.730,148.890
C05296=1154.524,404.228,-86.967,-176.164,9.728,148.889
C05297=1154.526,403.981,-86.930,-176.163,9.726,148.888
C05298=1154.530,403.734,-86.893,-176.163,9.725,148.888
C05299=1154.535,403.487,-86.856,-176.162,9.722,148.887
C05300=1154.539,403.239,-86.820,-176.161,9.721,148.886
C05301=1154.542,402.992,-86.783,-176.160,9.719,148.886
C05302=1154.546,402.745,-86.746,-176.159,9.717,148.885
C05303=1154.550,402.497,-86.709,-176.158,9.715,148.884
C05304=1154.554,402.250,-86.672,-176.157,9.713,148.883
C05305=1154.557,402.003,-86.636,-176.157,9.711,148.883
C05306=1154.561,401.756,-86.599,-176.155,9.709,148.882
C05307=1154.565,401.509,-86.562,-176.155,9.708,148.881
C05308=1154.569,401.262,-86.526,-176.154,9.705,148.880
C05309=1154.573,401.015,-86.489,-176.153,9.703,148.879
C05310=1154.576,400.766,-86.453,-176.152,9.701,148.879
C05311=1154.581,400.519,-86.416,-176.151,9.699,148.878
C05312=1154.585,400.272,-86.379,-176.151,9.697,148.877
C05313=1154.588,400.025,-86.343,-176.149,9.695,148.876
C05314=1154.592,399.778,-86.306,-176.148,9.693,148.876
C05315=1154.596,399.531,-86.269,-176.148,9.691,148.875
C05316=1154.600,399.283,-86.232,-176.147,9.688,148.874
C05317=1154.603,399.036,-86.196,-176.146,9.686,148.873
C05318=1154.607,398.789,-86.159,-176.145,9.685,148.873
C05319=1154.611,398.542,-86.122,-176.144,9.682,148.872
C05320=1154.615,398.294,-86.085,-176.143,9.680,148.871
C05321=1154.619,398.047,-86.049,-176.143,9.678,148.870
C05322=1154.623,397.800,-86.012,-176.142,9.676,148.869
C05323=1154.627,397.552,-85.975,-176.141,9.674,148.868
C05324=1154.631,397.305,-85.938,-176.140,9.672,148.868
C05325=1154.634,397.058,-85.902,-176.139,9.669,148.867
C05326=1154.638,396.811,-85.865,-176.138,9.667,148.866
C05327=1154.642,396.563,-85.829,-176.138,9.665,148.865
C05328=1154.646,396.316,-85.792,-176.137,9.662,148.865
C05329=1154.650,396.069,-85.755,-176.136,9.660,148.864
C05330=1154.654,395.822,-85.719,-176.135,9.657,148.863
C05331=1154.657,395.574,-85.681,-176.135,9.656,148.862
C05332=1154.661,395.327,-85.644,-176.134,9.654,148.861
C05333=1154.665,395.080,-85.608,-176.133,9.651,148.860
C05334=1154.669,394.832,-85.572,-176.132,9.649,148.860
C05335=1154.673,394.585,-85.535,-176.132,9.646,148.859
C05336=1154.677,394.338,-85.498,-176.131,9.644,148.858
C05337=1154.681,394.091,-85.462,-176.130,9.641,148.857
C05338=1154.684,393.843,-85.425,-176.130,9.638,148.856
C05339=1154.688,393.596,-85.388,-176.129,9.637,148.856
C05340=1154.692,393.349,-85.352,-176.128,9.634,148.855
C05341=1154.696,393.102,-85.315,-176.128,9.631,148.854
C05342=1154.700,392.855,-85.278,-176.127,9.629,148.853
C05343=1154.704,392.607,-85.242,-176.127,9.626,148.852
C05344=1154.708,392.360,-85.206,-176.126,9.623,148.851
C05345=1154.711,392.112,-85.168,-176.126,9.620,148.850
C05346=1154.715,391.865,-85.132,-176.124,9.618,148.850
C05347=1154.720,391.579,-85.089,-176.124,9.616,148.849
C05348=1154.724,391.293,-85.047,-176.124,9.612,148.848
C05349=1154.729,391.007,-85.005,-176.123,9.609,148.847
C05350=1154.733,390.721,-84.962,-176.122,9.606,148.846
C05351=1154.737,390.474,-84.925,-176.122,9.603,148.845
C05352=1154.740,390.226,-84.890,-176.122,9.600,148.844
C05353=1154.744,389.979,-84.853,-176.121,9.597,148.843
C05354=1154.749,389.732,-84.816,-176.121,9.595,148.842
C05355=1154.752,389.485,-84.780,-176.121,9.591,148.842
C05356=1154.755,389.237,-84.742,-176.121,9.588,148.841
C05357=1154.760,388.990,-84.706,-176.121,9.586,148.840
C05358=1154.763,388.742,-84.670,-176.120,9.583,148.839
C05359=1154.767,388.495,-84.633,-176.120,9.579,148.838
C05360=1154.771,388.248,-84.596,-176.120,9.577,148.837
C05361=1154.775,388.001,-84.560,-176.119,9.574,148.836
C05362=1154.779,387.754,-84.523,-176.120,9.570,148.836
C05363=1154.783,387.506,-84.487,-176.119,9.568,148.835
C05364=1154.787,387.259,-84.451,-176.120,9.564,148.834
C05365=1154.790,387.011,-84.413,-176.120,9.562,148.833
C05366=1154.794,386.764,-84.377,-176.120,9.558,148.832
C05367=1154.798,386.517,-84.340,-176.120,9.554,148.832
C05368=1154.802,386.269,-84.304,-176.120,9.552,148.831
C05369=1154.806,386.022,-84.267,-176.120,9.548,148.830
C05370=1154.809,385.775,-84.231,-176.120,9.545,148.829
C05371=1154.813,385.528,-84.194,-176.121,9.541,148.828
C05372=1154.817,385.281,-84.159,-176.121,9.538,148.828
C05373=1154.821,385.033,-84.122,-176.121,9.534,148.827
C05374=1154.825,384.786,-84.085,-176.122,9.531,148.826
C05375=1154.829,384.539,-84.049,-176.122,9.528,148.825
C05376=1154.833,384.292,-84.013,-176.123,9.524,148.824
C05377=1154.837,384.044,-83.975,-176.123,9.521,148.824
C05378=1154.840,383.797,-83.939,-176.124,9.517,148.823
C05379=1154.844,383.549,-83.903,-176.125,9.513,148.822
C05380=1154.848,383.302,-83.867,-176.125,9.510,148.821
C05381=1154.852,383.055,-83.830,-176.126,9.507,148.821
C05382=1154.855,382.807,-83.794,-176.127,9.503,148.820
C05383=1154.860,382.560,-83.757,-176.128,9.499,148.819
C05384=1154.864,382.313,-83.721,-176.129,9.495,148.818
C05385=1154.867,382.065,-83.685,-176.130,9.492,148.818
C05386=1154.871,381.818,-83.648,-176.131,9.488,148.817
C05387=1154.875,381.571,-83.613,-176.131,9.484,148.816
C05388=1154.879,381.324,-83.576,-176.133,9.480,148.816
C05389=1154.882,381.077,-83.539,-176.134,9.476,148.815
C05390=1154.887,380.829,-83.503,-176.134,9.473,148.814
C05391=1154.890,380.582,-83.467,-176.135,9.469,148.813
C05392=1154.895,380.334,-83.431,-176.137,9.465,148.813
C05393=1154.898,380.087,-83.395,-176.138,9.461,148.812
C05394=1154.902,379.840,-83.359,-176.139,9.457,148.811
C05395=1154.906,379.593,-83.322,-176.140,9.454,148.811
C05396=1154.910,379.345,-83.286,-176.142,9.450,148.810
C05397=1154.914,379.098,-83.250,-176.143,9.446,148.810
C05398=1154.918,378.850,-83.214,-176.145,9.442,148.809
C05399=1154.921,378.603,-83.177,-176.146,9.438,148.808
C05400=1154.926,378.355,-83.141,-176.148,9.434,148.808
C05401=1154.929,378.109,-83.105,-176.149,9.431,148.807
C05402=1154.933,377.861,-83.069,-176.151,9.427,148.806
C05403=1154.937,377.614,-83.033,-176.153,9.422,148.806
C05404=1154.941,377.366,-82.996,-176.154,9.418,148.805
C05405=1154.945,377.119,-82.961,-176.156,9.414,148.805
C05406=1154.949,376.871,-82.924,-176.157,9.410,148.804
C05407=1154.953,376.624,-82.889,-176.158,9.406,148.803
C05408=1154.956,376.377,-82.852,-176.160,9.403,148.803
C05409=1154.960,376.129,-82.816,-176.162,9.398,148.802
C05410=1154.964,375.882,-82.781,-176.164,9.394,148.802
C05411=1154.967,375.635,-82.744,-176.166,9.391,148.801
C05412=1154.972,375.387,-82.708,-176.168,9.386,148.800
C05413=1154.976,375.140,-82.673,-176.170,9.382,148.800
C05414=1154.980,374.893,-82.636,-176.171,9.378,148.799
C05415=1154.984,374.646,-82.601,-176.174,9.374,148.799
C05416=1154.987,374.398,-82.565,-176.175,9.370,148.798
C05417=1154.992,374.150,-82.529,-176.177,9.367,148.798
C05418=1154.995,373.903,-82.493,-176.179,9.362,148.797
C05419=1154.999,373.656,-82.457,-176.181,9.358,148.797
C05420=1155.003,373.408,-82.421,-176.183,9.354,148.796
C05421=1155.007,373.161,-82.385,-176.185,9.350,148.796
C05422=1155.011,372.913,-82.350,-176.187,9.346,148.795
C05423=1155.014,372.666,-82.314,-176.189,9.342,148.795
C05424=1155.019,372.419,-82.278,-176.191,9.338,148.794
C05425=1155.023,372.172,-82.242,-176.194,9.334,148.794
C05426=1155.026,371.924,-82.207,-176.195,9.330,148.793
C05427=1155.030,371.677,-82.171,-176.198,9.326,148.793
C05428=1155.034,371.429,-82.135,-176.200,9.322,148.793
C05429=1155.038,371.181,-82.099,-176.202,9.318,148.792
C05430=1155.042,370.934,-82.064,-176.204,9.314,148.792
C05431=1155.046,370.687,-82.029,-176.207,9.310,148.791
C05432=1155.050,370.439,-81.993,-176.209,9.306,148.791
C05433=1155.054,370.192,-81.957,-176.211,9.302,148.790
C05434=1155.058,369.944,-81.922,-176.213,9.298,148.790
C05435=1155.061,369.697,-81.886,-176.215,9.294,148.789
C05436=1155.066,369.450,-81.851,-176.218,9.290,148.789
C05437=1155.069,369.202,-81.815,-176.221,9.285,148.789
C05438=1155.074,368.954,-81.779,-176.223,9.282,148.788
C05439=1155.077,368.707,-81.744,-176.225,9.277,148.788
C05440=1155.081,368.459,-81.708,-176.227,9.274,148.787
C05441=1155.085,368.213,-81.673,-176.230,9.270,148.787
C05442=1155.089,367.965,-81.637,-176.232,9.265,148.787
C05443=1155.093,367.718,-81.602,-176.234,9.262,148.786
C05444=1155.096,367.470,-81.566,-176.237,9.258,148.786
C05445=1155.100,367.223,-81.531,-176.239,9.254,148.786
C05446=1155.105,366.975,-81.496,-176.241,9.250,148.785
C05447=1155.109,366.727,-81.460,-176.244,9.246,148.785
C05448=1155.113,366.480,-81.424,-176.246,9.242,148.784
C05449=1155.117,366.233,-81.389,-176.249,9.238,148.784
C05450=1155.120,365.986,-81.354,-176.252,9.234,148.784
C05451=1155.124,365.703,-81.314,-176.254,9.229,148.783
C05452=1155.129,365.420,-81.273,-176.257,9.225,148.783
C05453=1155.134,365.137,-81.232,-176.260,9.220,148.782
C05454=1155.138,364.854,-81.193,-176.263,9.216,148.782
C05455=1155.142,364.606,-81.158,-176.265,9.211,148.782
C05456=1155.146,364.359,-81.123,-176.268,9.208,148.781
C05457=1155.150,364.111,-81.088,-176.270,9.204,148.781
C05458=1155.154,363.864,-81.052,-176.272,9.200,148.781
C05459=1155.157,363.616,-81.017,-176.275,9.196,148.780
C05460=1155.162,363.369,-80.982,-176.278,9.192,148.780
C05461=1155.166,363.121,-80.947,-176.280,9.189,148.780
C05462=1155.169,362.874,-80.911,-176.283,9.184,148.779
C05463=1155.174,362.626,-80.877,-176.285,9.180,148.779
C05464=1155.178,362.379,-80.841,-176.287,9.176,148.779
C05465=1155.181,362.131,-80.806,-176.290,9.172,148.778
C05466=1155.185,361.884,-80.772,-176.293,9.168,148.778
C05467=1155.189,361.636,-80.737,-176.295,9.165,148.778
C05468=1155.193,361.389,-80.701,-176.298,9.161,148.777
C05469=1155.197,361.141,-80.667,-176.300,9.157,148.777
C05470=1155.201,360.894,-80.631,-176.303,9.153,148.777
C05471=1155.205,360.646,-80.597,-176.306,9.149,148.776
C05472=1155.209,360.399,-80.561,-176.307,9.145,148.776
C05473=1155.212,360.151,-80.527,-176.310,9.141,148.776
C05474=1155.217,359.904,-80.492,-176.313,9.138,148.776
C05475=1155.221,359.656,-80.457,-176.315,9.133,148.775
C05476=1155.225,359.409,-80.422,-176.318,9.129,148.775
C05477=1155.229,359.161,-80.387,-176.320,9.126,148.775
C05478=1155.232,358.913,-80.353,-176.323,9.122,148.774
C05479=1155.237,358.666,-80.318,-176.325,9.118,148.774
